   // UNICODE_TO_GBK[17326] := 16#6D0A;
   // UNICODE_TO_GBK[17327] := 16#9B96;
   // UNICODE_TO_GBK[17328] := 16#6D0B;
   // UNICODE_TO_GBK[17329] := 16#D1F3;
   // UNICODE_TO_GBK[17330] := 16#6D0C;
   // UNICODE_TO_GBK[17331] := 16#E4A3;
   // UNICODE_TO_GBK[17332] := 16#6D0D;
   // UNICODE_TO_GBK[17333] := 16#9B97;
   // UNICODE_TO_GBK[17334] := 16#6D0E;
   // UNICODE_TO_GBK[17335] := 16#E4A9;
   // UNICODE_TO_GBK[17336] := 16#6D0F;
   // UNICODE_TO_GBK[17337] := 16#9B98;
   // UNICODE_TO_GBK[17338] := 16#6D10;
   // UNICODE_TO_GBK[17339] := 16#9B99;
   // UNICODE_TO_GBK[17340] := 16#6D11;
   // UNICODE_TO_GBK[17341] := 16#9B9A;
   // UNICODE_TO_GBK[17342] := 16#6D12;
   // UNICODE_TO_GBK[17343] := 16#C8F7;
   // UNICODE_TO_GBK[17344] := 16#6D13;
   // UNICODE_TO_GBK[17345] := 16#9B9B;
   // UNICODE_TO_GBK[17346] := 16#6D14;
   // UNICODE_TO_GBK[17347] := 16#9B9C;
   // UNICODE_TO_GBK[17348] := 16#6D15;
   // UNICODE_TO_GBK[17349] := 16#9B9D;
   // UNICODE_TO_GBK[17350] := 16#6D16;
   // UNICODE_TO_GBK[17351] := 16#9B9E;
   // UNICODE_TO_GBK[17352] := 16#6D17;
   // UNICODE_TO_GBK[17353] := 16#CFB4;
   // UNICODE_TO_GBK[17354] := 16#6D18;
   // UNICODE_TO_GBK[17355] := 16#9B9F;
   // UNICODE_TO_GBK[17356] := 16#6D19;
   // UNICODE_TO_GBK[17357] := 16#E4A8;
   // UNICODE_TO_GBK[17358] := 16#6D1A;
   // UNICODE_TO_GBK[17359] := 16#E4AE;
   // UNICODE_TO_GBK[17360] := 16#6D1B;
   // UNICODE_TO_GBK[17361] := 16#C2E5;
   // UNICODE_TO_GBK[17362] := 16#6D1C;
   // UNICODE_TO_GBK[17363] := 16#9BA0;
   // UNICODE_TO_GBK[17364] := 16#6D1D;
   // UNICODE_TO_GBK[17365] := 16#9BA1;
   // UNICODE_TO_GBK[17366] := 16#6D1E;
   // UNICODE_TO_GBK[17367] := 16#B6B4;
   // UNICODE_TO_GBK[17368] := 16#6D1F;
   // UNICODE_TO_GBK[17369] := 16#9BA2;
   // UNICODE_TO_GBK[17370] := 16#6D20;
   // UNICODE_TO_GBK[17371] := 16#9BA3;
   // UNICODE_TO_GBK[17372] := 16#6D21;
   // UNICODE_TO_GBK[17373] := 16#9BA4;
   // UNICODE_TO_GBK[17374] := 16#6D22;
   // UNICODE_TO_GBK[17375] := 16#9BA5;
   // UNICODE_TO_GBK[17376] := 16#6D23;
   // UNICODE_TO_GBK[17377] := 16#9BA6;
   // UNICODE_TO_GBK[17378] := 16#6D24;
   // UNICODE_TO_GBK[17379] := 16#9BA7;
   // UNICODE_TO_GBK[17380] := 16#6D25;
   // UNICODE_TO_GBK[17381] := 16#BDF2;
   // UNICODE_TO_GBK[17382] := 16#6D26;
   // UNICODE_TO_GBK[17383] := 16#9BA8;
   // UNICODE_TO_GBK[17384] := 16#6D27;
   // UNICODE_TO_GBK[17385] := 16#E4A2;
   // UNICODE_TO_GBK[17386] := 16#6D28;
   // UNICODE_TO_GBK[17387] := 16#9BA9;
   // UNICODE_TO_GBK[17388] := 16#6D29;
   // UNICODE_TO_GBK[17389] := 16#9BAA;
   // UNICODE_TO_GBK[17390] := 16#6D2A;
   // UNICODE_TO_GBK[17391] := 16#BAE9;
   // UNICODE_TO_GBK[17392] := 16#6D2B;
   // UNICODE_TO_GBK[17393] := 16#E4AA;
   // UNICODE_TO_GBK[17394] := 16#6D2C;
   // UNICODE_TO_GBK[17395] := 16#9BAB;
   // UNICODE_TO_GBK[17396] := 16#6D2D;
   // UNICODE_TO_GBK[17397] := 16#9BAC;
   // UNICODE_TO_GBK[17398] := 16#6D2E;
   // UNICODE_TO_GBK[17399] := 16#E4AC;
   // UNICODE_TO_GBK[17400] := 16#6D2F;
   // UNICODE_TO_GBK[17401] := 16#9BAD;
   // UNICODE_TO_GBK[17402] := 16#6D30;
   // UNICODE_TO_GBK[17403] := 16#9BAE;
   // UNICODE_TO_GBK[17404] := 16#6D31;
   // UNICODE_TO_GBK[17405] := 16#B6FD;
   // UNICODE_TO_GBK[17406] := 16#6D32;
   // UNICODE_TO_GBK[17407] := 16#D6DE;
   // UNICODE_TO_GBK[17408] := 16#6D33;
   // UNICODE_TO_GBK[17409] := 16#E4B2;
   // UNICODE_TO_GBK[17410] := 16#6D34;
   // UNICODE_TO_GBK[17411] := 16#9BAF;
   // UNICODE_TO_GBK[17412] := 16#6D35;
   // UNICODE_TO_GBK[17413] := 16#E4AD;
   // UNICODE_TO_GBK[17414] := 16#6D36;
   // UNICODE_TO_GBK[17415] := 16#9BB0;
   // UNICODE_TO_GBK[17416] := 16#6D37;
   // UNICODE_TO_GBK[17417] := 16#9BB1;
   // UNICODE_TO_GBK[17418] := 16#6D38;
   // UNICODE_TO_GBK[17419] := 16#9BB2;
   // UNICODE_TO_GBK[17420] := 16#6D39;
   // UNICODE_TO_GBK[17421] := 16#E4A1;
   // UNICODE_TO_GBK[17422] := 16#6D3A;
   // UNICODE_TO_GBK[17423] := 16#9BB3;
   // UNICODE_TO_GBK[17424] := 16#6D3B;
   // UNICODE_TO_GBK[17425] := 16#BBEE;
   // UNICODE_TO_GBK[17426] := 16#6D3C;
   // UNICODE_TO_GBK[17427] := 16#CDDD;
   // UNICODE_TO_GBK[17428] := 16#6D3D;
   // UNICODE_TO_GBK[17429] := 16#C7A2;
   // UNICODE_TO_GBK[17430] := 16#6D3E;
   // UNICODE_TO_GBK[17431] := 16#C5C9;
   // UNICODE_TO_GBK[17432] := 16#6D3F;
   // UNICODE_TO_GBK[17433] := 16#9BB4;
   // UNICODE_TO_GBK[17434] := 16#6D40;
   // UNICODE_TO_GBK[17435] := 16#9BB5;
   // UNICODE_TO_GBK[17436] := 16#6D41;
   // UNICODE_TO_GBK[17437] := 16#C1F7;
   // UNICODE_TO_GBK[17438] := 16#6D42;
   // UNICODE_TO_GBK[17439] := 16#9BB6;
   // UNICODE_TO_GBK[17440] := 16#6D43;
   // UNICODE_TO_GBK[17441] := 16#E4A4;
   // UNICODE_TO_GBK[17442] := 16#6D44;
   // UNICODE_TO_GBK[17443] := 16#9BB7;
   // UNICODE_TO_GBK[17444] := 16#6D45;
   // UNICODE_TO_GBK[17445] := 16#C7B3;
   // UNICODE_TO_GBK[17446] := 16#6D46;
   // UNICODE_TO_GBK[17447] := 16#BDAC;
   // UNICODE_TO_GBK[17448] := 16#6D47;
   // UNICODE_TO_GBK[17449] := 16#BDBD;
   // UNICODE_TO_GBK[17450] := 16#6D48;
   // UNICODE_TO_GBK[17451] := 16#E4A5;
   // UNICODE_TO_GBK[17452] := 16#6D49;
   // UNICODE_TO_GBK[17453] := 16#9BB8;
   // UNICODE_TO_GBK[17454] := 16#6D4A;
   // UNICODE_TO_GBK[17455] := 16#D7C7;
   // UNICODE_TO_GBK[17456] := 16#6D4B;
   // UNICODE_TO_GBK[17457] := 16#B2E2;
   // UNICODE_TO_GBK[17458] := 16#6D4C;
   // UNICODE_TO_GBK[17459] := 16#9BB9;
   // UNICODE_TO_GBK[17460] := 16#6D4D;
   // UNICODE_TO_GBK[17461] := 16#E4AB;
   // UNICODE_TO_GBK[17462] := 16#6D4E;
   // UNICODE_TO_GBK[17463] := 16#BCC3;
   // UNICODE_TO_GBK[17464] := 16#6D4F;
   // UNICODE_TO_GBK[17465] := 16#E4AF;
   // UNICODE_TO_GBK[17466] := 16#6D50;
   // UNICODE_TO_GBK[17467] := 16#9BBA;
   // UNICODE_TO_GBK[17468] := 16#6D51;
   // UNICODE_TO_GBK[17469] := 16#BBEB;
   // UNICODE_TO_GBK[17470] := 16#6D52;
   // UNICODE_TO_GBK[17471] := 16#E4B0;
   // UNICODE_TO_GBK[17472] := 16#6D53;
   // UNICODE_TO_GBK[17473] := 16#C5A8;
   // UNICODE_TO_GBK[17474] := 16#6D54;
   // UNICODE_TO_GBK[17475] := 16#E4B1;
   // UNICODE_TO_GBK[17476] := 16#6D55;
   // UNICODE_TO_GBK[17477] := 16#9BBB;
   // UNICODE_TO_GBK[17478] := 16#6D56;
   // UNICODE_TO_GBK[17479] := 16#9BBC;
   // UNICODE_TO_GBK[17480] := 16#6D57;
   // UNICODE_TO_GBK[17481] := 16#9BBD;
   // UNICODE_TO_GBK[17482] := 16#6D58;
   // UNICODE_TO_GBK[17483] := 16#9BBE;
   // UNICODE_TO_GBK[17484] := 16#6D59;
   // UNICODE_TO_GBK[17485] := 16#D5E3;
   // UNICODE_TO_GBK[17486] := 16#6D5A;
   // UNICODE_TO_GBK[17487] := 16#BFA3;
   // UNICODE_TO_GBK[17488] := 16#6D5B;
   // UNICODE_TO_GBK[17489] := 16#9BBF;
   // UNICODE_TO_GBK[17490] := 16#6D5C;
   // UNICODE_TO_GBK[17491] := 16#E4BA;
   // UNICODE_TO_GBK[17492] := 16#6D5D;
   // UNICODE_TO_GBK[17493] := 16#9BC0;
   // UNICODE_TO_GBK[17494] := 16#6D5E;
   // UNICODE_TO_GBK[17495] := 16#E4B7;
   // UNICODE_TO_GBK[17496] := 16#6D5F;
   // UNICODE_TO_GBK[17497] := 16#9BC1;
   // UNICODE_TO_GBK[17498] := 16#6D60;
   // UNICODE_TO_GBK[17499] := 16#E4BB;
   // UNICODE_TO_GBK[17500] := 16#6D61;
   // UNICODE_TO_GBK[17501] := 16#9BC2;
   // UNICODE_TO_GBK[17502] := 16#6D62;
   // UNICODE_TO_GBK[17503] := 16#9BC3;
   // UNICODE_TO_GBK[17504] := 16#6D63;
   // UNICODE_TO_GBK[17505] := 16#E4BD;
   // UNICODE_TO_GBK[17506] := 16#6D64;
   // UNICODE_TO_GBK[17507] := 16#9BC4;
   // UNICODE_TO_GBK[17508] := 16#6D65;
   // UNICODE_TO_GBK[17509] := 16#9BC5;
   // UNICODE_TO_GBK[17510] := 16#6D66;
   // UNICODE_TO_GBK[17511] := 16#C6D6;
   // UNICODE_TO_GBK[17512] := 16#6D67;
   // UNICODE_TO_GBK[17513] := 16#9BC6;
   // UNICODE_TO_GBK[17514] := 16#6D68;
   // UNICODE_TO_GBK[17515] := 16#9BC7;
   // UNICODE_TO_GBK[17516] := 16#6D69;
   // UNICODE_TO_GBK[17517] := 16#BAC6;
   // UNICODE_TO_GBK[17518] := 16#6D6A;
   // UNICODE_TO_GBK[17519] := 16#C0CB;
   // UNICODE_TO_GBK[17520] := 16#6D6B;
   // UNICODE_TO_GBK[17521] := 16#9BC8;
   // UNICODE_TO_GBK[17522] := 16#6D6C;
   // UNICODE_TO_GBK[17523] := 16#9BC9;
   // UNICODE_TO_GBK[17524] := 16#6D6D;
   // UNICODE_TO_GBK[17525] := 16#9BCA;
   // UNICODE_TO_GBK[17526] := 16#6D6E;
   // UNICODE_TO_GBK[17527] := 16#B8A1;
   // UNICODE_TO_GBK[17528] := 16#6D6F;
   // UNICODE_TO_GBK[17529] := 16#E4B4;
   // UNICODE_TO_GBK[17530] := 16#6D70;
   // UNICODE_TO_GBK[17531] := 16#9BCB;
   // UNICODE_TO_GBK[17532] := 16#6D71;
   // UNICODE_TO_GBK[17533] := 16#9BCC;
   // UNICODE_TO_GBK[17534] := 16#6D72;
   // UNICODE_TO_GBK[17535] := 16#9BCD;
   // UNICODE_TO_GBK[17536] := 16#6D73;
   // UNICODE_TO_GBK[17537] := 16#9BCE;
   // UNICODE_TO_GBK[17538] := 16#6D74;
   // UNICODE_TO_GBK[17539] := 16#D4A1;
   // UNICODE_TO_GBK[17540] := 16#6D75;
   // UNICODE_TO_GBK[17541] := 16#9BCF;
   // UNICODE_TO_GBK[17542] := 16#6D76;
   // UNICODE_TO_GBK[17543] := 16#9BD0;
   // UNICODE_TO_GBK[17544] := 16#6D77;
   // UNICODE_TO_GBK[17545] := 16#BAA3;
   // UNICODE_TO_GBK[17546] := 16#6D78;
   // UNICODE_TO_GBK[17547] := 16#BDFE;
   // UNICODE_TO_GBK[17548] := 16#6D79;
   // UNICODE_TO_GBK[17549] := 16#9BD1;
   // UNICODE_TO_GBK[17550] := 16#6D7A;
   // UNICODE_TO_GBK[17551] := 16#9BD2;
   // UNICODE_TO_GBK[17552] := 16#6D7B;
   // UNICODE_TO_GBK[17553] := 16#9BD3;
   // UNICODE_TO_GBK[17554] := 16#6D7C;
   // UNICODE_TO_GBK[17555] := 16#E4BC;
   // UNICODE_TO_GBK[17556] := 16#6D7D;
   // UNICODE_TO_GBK[17557] := 16#9BD4;
   // UNICODE_TO_GBK[17558] := 16#6D7E;
   // UNICODE_TO_GBK[17559] := 16#9BD5;
   // UNICODE_TO_GBK[17560] := 16#6D7F;
   // UNICODE_TO_GBK[17561] := 16#9BD6;
   // UNICODE_TO_GBK[17562] := 16#6D80;
   // UNICODE_TO_GBK[17563] := 16#9BD7;
   // UNICODE_TO_GBK[17564] := 16#6D81;
   // UNICODE_TO_GBK[17565] := 16#9BD8;
   // UNICODE_TO_GBK[17566] := 16#6D82;
   // UNICODE_TO_GBK[17567] := 16#CDBF;
   // UNICODE_TO_GBK[17568] := 16#6D83;
   // UNICODE_TO_GBK[17569] := 16#9BD9;
   // UNICODE_TO_GBK[17570] := 16#6D84;
   // UNICODE_TO_GBK[17571] := 16#9BDA;
   // UNICODE_TO_GBK[17572] := 16#6D85;
   // UNICODE_TO_GBK[17573] := 16#C4F9;
   // UNICODE_TO_GBK[17574] := 16#6D86;
   // UNICODE_TO_GBK[17575] := 16#9BDB;
   // UNICODE_TO_GBK[17576] := 16#6D87;
   // UNICODE_TO_GBK[17577] := 16#9BDC;
   // UNICODE_TO_GBK[17578] := 16#6D88;
   // UNICODE_TO_GBK[17579] := 16#CFFB;
   // UNICODE_TO_GBK[17580] := 16#6D89;
   // UNICODE_TO_GBK[17581] := 16#C9E6;
   // UNICODE_TO_GBK[17582] := 16#6D8A;
   // UNICODE_TO_GBK[17583] := 16#9BDD;
   // UNICODE_TO_GBK[17584] := 16#6D8B;
   // UNICODE_TO_GBK[17585] := 16#9BDE;
   // UNICODE_TO_GBK[17586] := 16#6D8C;
   // UNICODE_TO_GBK[17587] := 16#D3BF;
   // UNICODE_TO_GBK[17588] := 16#6D8D;
   // UNICODE_TO_GBK[17589] := 16#9BDF;
   // UNICODE_TO_GBK[17590] := 16#6D8E;
   // UNICODE_TO_GBK[17591] := 16#CFD1;
   // UNICODE_TO_GBK[17592] := 16#6D8F;
   // UNICODE_TO_GBK[17593] := 16#9BE0;
   // UNICODE_TO_GBK[17594] := 16#6D90;
   // UNICODE_TO_GBK[17595] := 16#9BE1;
   // UNICODE_TO_GBK[17596] := 16#6D91;
   // UNICODE_TO_GBK[17597] := 16#E4B3;
   // UNICODE_TO_GBK[17598] := 16#6D92;
   // UNICODE_TO_GBK[17599] := 16#9BE2;
   // UNICODE_TO_GBK[17600] := 16#6D93;
   // UNICODE_TO_GBK[17601] := 16#E4B8;
   // UNICODE_TO_GBK[17602] := 16#6D94;
   // UNICODE_TO_GBK[17603] := 16#E4B9;
   // UNICODE_TO_GBK[17604] := 16#6D95;
   // UNICODE_TO_GBK[17605] := 16#CCE9;
   // UNICODE_TO_GBK[17606] := 16#6D96;
   // UNICODE_TO_GBK[17607] := 16#9BE3;
   // UNICODE_TO_GBK[17608] := 16#6D97;
   // UNICODE_TO_GBK[17609] := 16#9BE4;
   // UNICODE_TO_GBK[17610] := 16#6D98;
   // UNICODE_TO_GBK[17611] := 16#9BE5;
   // UNICODE_TO_GBK[17612] := 16#6D99;
   // UNICODE_TO_GBK[17613] := 16#9BE6;
   // UNICODE_TO_GBK[17614] := 16#6D9A;
   // UNICODE_TO_GBK[17615] := 16#9BE7;
   // UNICODE_TO_GBK[17616] := 16#6D9B;
   // UNICODE_TO_GBK[17617] := 16#CCCE;
   // UNICODE_TO_GBK[17618] := 16#6D9C;
   // UNICODE_TO_GBK[17619] := 16#9BE8;
   // UNICODE_TO_GBK[17620] := 16#6D9D;
   // UNICODE_TO_GBK[17621] := 16#C0D4;
   // UNICODE_TO_GBK[17622] := 16#6D9E;
   // UNICODE_TO_GBK[17623] := 16#E4B5;
   // UNICODE_TO_GBK[17624] := 16#6D9F;
   // UNICODE_TO_GBK[17625] := 16#C1B0;
   // UNICODE_TO_GBK[17626] := 16#6DA0;
   // UNICODE_TO_GBK[17627] := 16#E4B6;
   // UNICODE_TO_GBK[17628] := 16#6DA1;
   // UNICODE_TO_GBK[17629] := 16#CED0;
   // UNICODE_TO_GBK[17630] := 16#6DA2;
   // UNICODE_TO_GBK[17631] := 16#9BE9;
   // UNICODE_TO_GBK[17632] := 16#6DA3;
   // UNICODE_TO_GBK[17633] := 16#BBC1;
   // UNICODE_TO_GBK[17634] := 16#6DA4;
   // UNICODE_TO_GBK[17635] := 16#B5D3;
   // UNICODE_TO_GBK[17636] := 16#6DA5;
   // UNICODE_TO_GBK[17637] := 16#9BEA;
   // UNICODE_TO_GBK[17638] := 16#6DA6;
   // UNICODE_TO_GBK[17639] := 16#C8F3;
   // UNICODE_TO_GBK[17640] := 16#6DA7;
   // UNICODE_TO_GBK[17641] := 16#BDA7;
   // UNICODE_TO_GBK[17642] := 16#6DA8;
   // UNICODE_TO_GBK[17643] := 16#D5C7;
   // UNICODE_TO_GBK[17644] := 16#6DA9;
   // UNICODE_TO_GBK[17645] := 16#C9AC;
   // UNICODE_TO_GBK[17646] := 16#6DAA;
   // UNICODE_TO_GBK[17647] := 16#B8A2;
   // UNICODE_TO_GBK[17648] := 16#6DAB;
   // UNICODE_TO_GBK[17649] := 16#E4CA;
   // UNICODE_TO_GBK[17650] := 16#6DAC;
   // UNICODE_TO_GBK[17651] := 16#9BEB;
   // UNICODE_TO_GBK[17652] := 16#6DAD;
   // UNICODE_TO_GBK[17653] := 16#9BEC;
   // UNICODE_TO_GBK[17654] := 16#6DAE;
   // UNICODE_TO_GBK[17655] := 16#E4CC;
   // UNICODE_TO_GBK[17656] := 16#6DAF;
   // UNICODE_TO_GBK[17657] := 16#D1C4;
   // UNICODE_TO_GBK[17658] := 16#6DB0;
   // UNICODE_TO_GBK[17659] := 16#9BED;
   // UNICODE_TO_GBK[17660] := 16#6DB1;
   // UNICODE_TO_GBK[17661] := 16#9BEE;
   // UNICODE_TO_GBK[17662] := 16#6DB2;
   // UNICODE_TO_GBK[17663] := 16#D2BA;
   // UNICODE_TO_GBK[17664] := 16#6DB3;
   // UNICODE_TO_GBK[17665] := 16#9BEF;
   // UNICODE_TO_GBK[17666] := 16#6DB4;
   // UNICODE_TO_GBK[17667] := 16#9BF0;
   // UNICODE_TO_GBK[17668] := 16#6DB5;
   // UNICODE_TO_GBK[17669] := 16#BAAD;
   // UNICODE_TO_GBK[17670] := 16#6DB6;
   // UNICODE_TO_GBK[17671] := 16#9BF1;
   // UNICODE_TO_GBK[17672] := 16#6DB7;
   // UNICODE_TO_GBK[17673] := 16#9BF2;
   // UNICODE_TO_GBK[17674] := 16#6DB8;
   // UNICODE_TO_GBK[17675] := 16#BAD4;
   // UNICODE_TO_GBK[17676] := 16#6DB9;
   // UNICODE_TO_GBK[17677] := 16#9BF3;
   // UNICODE_TO_GBK[17678] := 16#6DBA;
   // UNICODE_TO_GBK[17679] := 16#9BF4;
   // UNICODE_TO_GBK[17680] := 16#6DBB;
   // UNICODE_TO_GBK[17681] := 16#9BF5;
   // UNICODE_TO_GBK[17682] := 16#6DBC;
   // UNICODE_TO_GBK[17683] := 16#9BF6;
   // UNICODE_TO_GBK[17684] := 16#6DBD;
   // UNICODE_TO_GBK[17685] := 16#9BF7;
   // UNICODE_TO_GBK[17686] := 16#6DBE;
   // UNICODE_TO_GBK[17687] := 16#9BF8;
   // UNICODE_TO_GBK[17688] := 16#6DBF;
   // UNICODE_TO_GBK[17689] := 16#E4C3;
   // UNICODE_TO_GBK[17690] := 16#6DC0;
   // UNICODE_TO_GBK[17691] := 16#B5ED;
   // UNICODE_TO_GBK[17692] := 16#6DC1;
   // UNICODE_TO_GBK[17693] := 16#9BF9;
   // UNICODE_TO_GBK[17694] := 16#6DC2;
   // UNICODE_TO_GBK[17695] := 16#9BFA;
   // UNICODE_TO_GBK[17696] := 16#6DC3;
   // UNICODE_TO_GBK[17697] := 16#9BFB;
   // UNICODE_TO_GBK[17698] := 16#6DC4;
   // UNICODE_TO_GBK[17699] := 16#D7CD;
   // UNICODE_TO_GBK[17700] := 16#6DC5;
   // UNICODE_TO_GBK[17701] := 16#E4C0;
   // UNICODE_TO_GBK[17702] := 16#6DC6;
   // UNICODE_TO_GBK[17703] := 16#CFFD;
   // UNICODE_TO_GBK[17704] := 16#6DC7;
   // UNICODE_TO_GBK[17705] := 16#E4BF;
   // UNICODE_TO_GBK[17706] := 16#6DC8;
   // UNICODE_TO_GBK[17707] := 16#9BFC;
   // UNICODE_TO_GBK[17708] := 16#6DC9;
   // UNICODE_TO_GBK[17709] := 16#9BFD;
   // UNICODE_TO_GBK[17710] := 16#6DCA;
   // UNICODE_TO_GBK[17711] := 16#9BFE;
   // UNICODE_TO_GBK[17712] := 16#6DCB;
   // UNICODE_TO_GBK[17713] := 16#C1DC;
   // UNICODE_TO_GBK[17714] := 16#6DCC;
   // UNICODE_TO_GBK[17715] := 16#CCCA;
   // UNICODE_TO_GBK[17716] := 16#6DCD;
   // UNICODE_TO_GBK[17717] := 16#9C40;
   // UNICODE_TO_GBK[17718] := 16#6DCE;
   // UNICODE_TO_GBK[17719] := 16#9C41;
   // UNICODE_TO_GBK[17720] := 16#6DCF;
   // UNICODE_TO_GBK[17721] := 16#9C42;
   // UNICODE_TO_GBK[17722] := 16#6DD0;
   // UNICODE_TO_GBK[17723] := 16#9C43;
   // UNICODE_TO_GBK[17724] := 16#6DD1;
   // UNICODE_TO_GBK[17725] := 16#CAE7;
   // UNICODE_TO_GBK[17726] := 16#6DD2;
   // UNICODE_TO_GBK[17727] := 16#9C44;
   // UNICODE_TO_GBK[17728] := 16#6DD3;
   // UNICODE_TO_GBK[17729] := 16#9C45;
   // UNICODE_TO_GBK[17730] := 16#6DD4;
   // UNICODE_TO_GBK[17731] := 16#9C46;
   // UNICODE_TO_GBK[17732] := 16#6DD5;
   // UNICODE_TO_GBK[17733] := 16#9C47;
   // UNICODE_TO_GBK[17734] := 16#6DD6;
   // UNICODE_TO_GBK[17735] := 16#C4D7;
   // UNICODE_TO_GBK[17736] := 16#6DD7;
   // UNICODE_TO_GBK[17737] := 16#9C48;
   // UNICODE_TO_GBK[17738] := 16#6DD8;
   // UNICODE_TO_GBK[17739] := 16#CCD4;
   // UNICODE_TO_GBK[17740] := 16#6DD9;
   // UNICODE_TO_GBK[17741] := 16#E4C8;
   // UNICODE_TO_GBK[17742] := 16#6DDA;
   // UNICODE_TO_GBK[17743] := 16#9C49;
   // UNICODE_TO_GBK[17744] := 16#6DDB;
   // UNICODE_TO_GBK[17745] := 16#9C4A;
   // UNICODE_TO_GBK[17746] := 16#6DDC;
   // UNICODE_TO_GBK[17747] := 16#9C4B;
   // UNICODE_TO_GBK[17748] := 16#6DDD;
   // UNICODE_TO_GBK[17749] := 16#E4C7;
   // UNICODE_TO_GBK[17750] := 16#6DDE;
   // UNICODE_TO_GBK[17751] := 16#E4C1;
   // UNICODE_TO_GBK[17752] := 16#6DDF;
   // UNICODE_TO_GBK[17753] := 16#9C4C;
   // UNICODE_TO_GBK[17754] := 16#6DE0;
   // UNICODE_TO_GBK[17755] := 16#E4C4;
   // UNICODE_TO_GBK[17756] := 16#6DE1;
   // UNICODE_TO_GBK[17757] := 16#B5AD;
   // UNICODE_TO_GBK[17758] := 16#6DE2;
   // UNICODE_TO_GBK[17759] := 16#9C4D;
   // UNICODE_TO_GBK[17760] := 16#6DE3;
   // UNICODE_TO_GBK[17761] := 16#9C4E;
   // UNICODE_TO_GBK[17762] := 16#6DE4;
   // UNICODE_TO_GBK[17763] := 16#D3D9;
   // UNICODE_TO_GBK[17764] := 16#6DE5;
   // UNICODE_TO_GBK[17765] := 16#9C4F;
   // UNICODE_TO_GBK[17766] := 16#6DE6;
   // UNICODE_TO_GBK[17767] := 16#E4C6;
   // UNICODE_TO_GBK[17768] := 16#6DE7;
   // UNICODE_TO_GBK[17769] := 16#9C50;
   // UNICODE_TO_GBK[17770] := 16#6DE8;
   // UNICODE_TO_GBK[17771] := 16#9C51;
   // UNICODE_TO_GBK[17772] := 16#6DE9;
   // UNICODE_TO_GBK[17773] := 16#9C52;
   // UNICODE_TO_GBK[17774] := 16#6DEA;
   // UNICODE_TO_GBK[17775] := 16#9C53;
   // UNICODE_TO_GBK[17776] := 16#6DEB;
   // UNICODE_TO_GBK[17777] := 16#D2F9;
   // UNICODE_TO_GBK[17778] := 16#6DEC;
   // UNICODE_TO_GBK[17779] := 16#B4E3;
   // UNICODE_TO_GBK[17780] := 16#6DED;
   // UNICODE_TO_GBK[17781] := 16#9C54;
   // UNICODE_TO_GBK[17782] := 16#6DEE;
   // UNICODE_TO_GBK[17783] := 16#BBB4;
   // UNICODE_TO_GBK[17784] := 16#6DEF;
   // UNICODE_TO_GBK[17785] := 16#9C55;
   // UNICODE_TO_GBK[17786] := 16#6DF0;
   // UNICODE_TO_GBK[17787] := 16#9C56;
   // UNICODE_TO_GBK[17788] := 16#6DF1;
   // UNICODE_TO_GBK[17789] := 16#C9EE;
   // UNICODE_TO_GBK[17790] := 16#6DF2;
   // UNICODE_TO_GBK[17791] := 16#9C57;
   // UNICODE_TO_GBK[17792] := 16#6DF3;
   // UNICODE_TO_GBK[17793] := 16#B4BE;
   // UNICODE_TO_GBK[17794] := 16#6DF4;
   // UNICODE_TO_GBK[17795] := 16#9C58;
   // UNICODE_TO_GBK[17796] := 16#6DF5;
   // UNICODE_TO_GBK[17797] := 16#9C59;
   // UNICODE_TO_GBK[17798] := 16#6DF6;
   // UNICODE_TO_GBK[17799] := 16#9C5A;
   // UNICODE_TO_GBK[17800] := 16#6DF7;
   // UNICODE_TO_GBK[17801] := 16#BBEC;
   // UNICODE_TO_GBK[17802] := 16#6DF8;
   // UNICODE_TO_GBK[17803] := 16#9C5B;
   // UNICODE_TO_GBK[17804] := 16#6DF9;
   // UNICODE_TO_GBK[17805] := 16#D1CD;
   // UNICODE_TO_GBK[17806] := 16#6DFA;
   // UNICODE_TO_GBK[17807] := 16#9C5C;
   // UNICODE_TO_GBK[17808] := 16#6DFB;
   // UNICODE_TO_GBK[17809] := 16#CCED;
   // UNICODE_TO_GBK[17810] := 16#6DFC;
   // UNICODE_TO_GBK[17811] := 16#EDB5;
   // UNICODE_TO_GBK[17812] := 16#6DFD;
   // UNICODE_TO_GBK[17813] := 16#9C5D;
   // UNICODE_TO_GBK[17814] := 16#6DFE;
   // UNICODE_TO_GBK[17815] := 16#9C5E;
   // UNICODE_TO_GBK[17816] := 16#6DFF;
   // UNICODE_TO_GBK[17817] := 16#9C5F;
   // UNICODE_TO_GBK[17818] := 16#6E00;
   // UNICODE_TO_GBK[17819] := 16#9C60;
   // UNICODE_TO_GBK[17820] := 16#6E01;
   // UNICODE_TO_GBK[17821] := 16#9C61;
   // UNICODE_TO_GBK[17822] := 16#6E02;
   // UNICODE_TO_GBK[17823] := 16#9C62;
   // UNICODE_TO_GBK[17824] := 16#6E03;
   // UNICODE_TO_GBK[17825] := 16#9C63;
   // UNICODE_TO_GBK[17826] := 16#6E04;
   // UNICODE_TO_GBK[17827] := 16#9C64;
   // UNICODE_TO_GBK[17828] := 16#6E05;
   // UNICODE_TO_GBK[17829] := 16#C7E5;
   // UNICODE_TO_GBK[17830] := 16#6E06;
   // UNICODE_TO_GBK[17831] := 16#9C65;
   // UNICODE_TO_GBK[17832] := 16#6E07;
   // UNICODE_TO_GBK[17833] := 16#9C66;
   // UNICODE_TO_GBK[17834] := 16#6E08;
   // UNICODE_TO_GBK[17835] := 16#9C67;
   // UNICODE_TO_GBK[17836] := 16#6E09;
   // UNICODE_TO_GBK[17837] := 16#9C68;
   // UNICODE_TO_GBK[17838] := 16#6E0A;
   // UNICODE_TO_GBK[17839] := 16#D4A8;
   // UNICODE_TO_GBK[17840] := 16#6E0B;
   // UNICODE_TO_GBK[17841] := 16#9C69;
   // UNICODE_TO_GBK[17842] := 16#6E0C;
   // UNICODE_TO_GBK[17843] := 16#E4CB;
   // UNICODE_TO_GBK[17844] := 16#6E0D;
   // UNICODE_TO_GBK[17845] := 16#D7D5;
   // UNICODE_TO_GBK[17846] := 16#6E0E;
   // UNICODE_TO_GBK[17847] := 16#E4C2;
   // UNICODE_TO_GBK[17848] := 16#6E0F;
   // UNICODE_TO_GBK[17849] := 16#9C6A;
   // UNICODE_TO_GBK[17850] := 16#6E10;
   // UNICODE_TO_GBK[17851] := 16#BDA5;
   // UNICODE_TO_GBK[17852] := 16#6E11;
   // UNICODE_TO_GBK[17853] := 16#E4C5;
   // UNICODE_TO_GBK[17854] := 16#6E12;
   // UNICODE_TO_GBK[17855] := 16#9C6B;
   // UNICODE_TO_GBK[17856] := 16#6E13;
   // UNICODE_TO_GBK[17857] := 16#9C6C;
   // UNICODE_TO_GBK[17858] := 16#6E14;
   // UNICODE_TO_GBK[17859] := 16#D3E6;
   // UNICODE_TO_GBK[17860] := 16#6E15;
   // UNICODE_TO_GBK[17861] := 16#9C6D;
   // UNICODE_TO_GBK[17862] := 16#6E16;
   // UNICODE_TO_GBK[17863] := 16#E4C9;
   // UNICODE_TO_GBK[17864] := 16#6E17;
   // UNICODE_TO_GBK[17865] := 16#C9F8;
   // UNICODE_TO_GBK[17866] := 16#6E18;
   // UNICODE_TO_GBK[17867] := 16#9C6E;
   // UNICODE_TO_GBK[17868] := 16#6E19;
   // UNICODE_TO_GBK[17869] := 16#9C6F;
   // UNICODE_TO_GBK[17870] := 16#6E1A;
   // UNICODE_TO_GBK[17871] := 16#E4BE;
   // UNICODE_TO_GBK[17872] := 16#6E1B;
   // UNICODE_TO_GBK[17873] := 16#9C70;
   // UNICODE_TO_GBK[17874] := 16#6E1C;
   // UNICODE_TO_GBK[17875] := 16#9C71;
   // UNICODE_TO_GBK[17876] := 16#6E1D;
   // UNICODE_TO_GBK[17877] := 16#D3E5;
   // UNICODE_TO_GBK[17878] := 16#6E1E;
   // UNICODE_TO_GBK[17879] := 16#9C72;
   // UNICODE_TO_GBK[17880] := 16#6E1F;
   // UNICODE_TO_GBK[17881] := 16#9C73;
   // UNICODE_TO_GBK[17882] := 16#6E20;
   // UNICODE_TO_GBK[17883] := 16#C7FE;
   // UNICODE_TO_GBK[17884] := 16#6E21;
   // UNICODE_TO_GBK[17885] := 16#B6C9;
   // UNICODE_TO_GBK[17886] := 16#6E22;
   // UNICODE_TO_GBK[17887] := 16#9C74;
   // UNICODE_TO_GBK[17888] := 16#6E23;
   // UNICODE_TO_GBK[17889] := 16#D4FC;
   // UNICODE_TO_GBK[17890] := 16#6E24;
   // UNICODE_TO_GBK[17891] := 16#B2B3;
   // UNICODE_TO_GBK[17892] := 16#6E25;
   // UNICODE_TO_GBK[17893] := 16#E4D7;
   // UNICODE_TO_GBK[17894] := 16#6E26;
   // UNICODE_TO_GBK[17895] := 16#9C75;
   // UNICODE_TO_GBK[17896] := 16#6E27;
   // UNICODE_TO_GBK[17897] := 16#9C76;
   // UNICODE_TO_GBK[17898] := 16#6E28;
   // UNICODE_TO_GBK[17899] := 16#9C77;
   // UNICODE_TO_GBK[17900] := 16#6E29;
   // UNICODE_TO_GBK[17901] := 16#CEC2;
   // UNICODE_TO_GBK[17902] := 16#6E2A;
   // UNICODE_TO_GBK[17903] := 16#9C78;
   // UNICODE_TO_GBK[17904] := 16#6E2B;
   // UNICODE_TO_GBK[17905] := 16#E4CD;
   // UNICODE_TO_GBK[17906] := 16#6E2C;
   // UNICODE_TO_GBK[17907] := 16#9C79;
   // UNICODE_TO_GBK[17908] := 16#6E2D;
   // UNICODE_TO_GBK[17909] := 16#CEBC;
   // UNICODE_TO_GBK[17910] := 16#6E2E;
   // UNICODE_TO_GBK[17911] := 16#9C7A;
   // UNICODE_TO_GBK[17912] := 16#6E2F;
   // UNICODE_TO_GBK[17913] := 16#B8DB;
   // UNICODE_TO_GBK[17914] := 16#6E30;
   // UNICODE_TO_GBK[17915] := 16#9C7B;
   // UNICODE_TO_GBK[17916] := 16#6E31;
   // UNICODE_TO_GBK[17917] := 16#9C7C;
   // UNICODE_TO_GBK[17918] := 16#6E32;
   // UNICODE_TO_GBK[17919] := 16#E4D6;
   // UNICODE_TO_GBK[17920] := 16#6E33;
   // UNICODE_TO_GBK[17921] := 16#9C7D;
   // UNICODE_TO_GBK[17922] := 16#6E34;
   // UNICODE_TO_GBK[17923] := 16#BFCA;
   // UNICODE_TO_GBK[17924] := 16#6E35;
   // UNICODE_TO_GBK[17925] := 16#9C7E;
   // UNICODE_TO_GBK[17926] := 16#6E36;
   // UNICODE_TO_GBK[17927] := 16#9C80;
   // UNICODE_TO_GBK[17928] := 16#6E37;
   // UNICODE_TO_GBK[17929] := 16#9C81;
   // UNICODE_TO_GBK[17930] := 16#6E38;
   // UNICODE_TO_GBK[17931] := 16#D3CE;
   // UNICODE_TO_GBK[17932] := 16#6E39;
   // UNICODE_TO_GBK[17933] := 16#9C82;
   // UNICODE_TO_GBK[17934] := 16#6E3A;
   // UNICODE_TO_GBK[17935] := 16#C3EC;
   // UNICODE_TO_GBK[17936] := 16#6E3B;
   // UNICODE_TO_GBK[17937] := 16#9C83;
   // UNICODE_TO_GBK[17938] := 16#6E3C;
   // UNICODE_TO_GBK[17939] := 16#9C84;
   // UNICODE_TO_GBK[17940] := 16#6E3D;
   // UNICODE_TO_GBK[17941] := 16#9C85;
   // UNICODE_TO_GBK[17942] := 16#6E3E;
   // UNICODE_TO_GBK[17943] := 16#9C86;
   // UNICODE_TO_GBK[17944] := 16#6E3F;
   // UNICODE_TO_GBK[17945] := 16#9C87;
   // UNICODE_TO_GBK[17946] := 16#6E40;
   // UNICODE_TO_GBK[17947] := 16#9C88;
   // UNICODE_TO_GBK[17948] := 16#6E41;
   // UNICODE_TO_GBK[17949] := 16#9C89;
   // UNICODE_TO_GBK[17950] := 16#6E42;
   // UNICODE_TO_GBK[17951] := 16#9C8A;
   // UNICODE_TO_GBK[17952] := 16#6E43;
   // UNICODE_TO_GBK[17953] := 16#C5C8;
   // UNICODE_TO_GBK[17954] := 16#6E44;
   // UNICODE_TO_GBK[17955] := 16#E4D8;
   // UNICODE_TO_GBK[17956] := 16#6E45;
   // UNICODE_TO_GBK[17957] := 16#9C8B;
   // UNICODE_TO_GBK[17958] := 16#6E46;
   // UNICODE_TO_GBK[17959] := 16#9C8C;
   // UNICODE_TO_GBK[17960] := 16#6E47;
   // UNICODE_TO_GBK[17961] := 16#9C8D;
   // UNICODE_TO_GBK[17962] := 16#6E48;
   // UNICODE_TO_GBK[17963] := 16#9C8E;
   // UNICODE_TO_GBK[17964] := 16#6E49;
   // UNICODE_TO_GBK[17965] := 16#9C8F;
   // UNICODE_TO_GBK[17966] := 16#6E4A;
   // UNICODE_TO_GBK[17967] := 16#9C90;
   // UNICODE_TO_GBK[17968] := 16#6E4B;
   // UNICODE_TO_GBK[17969] := 16#9C91;
   // UNICODE_TO_GBK[17970] := 16#6E4C;
   // UNICODE_TO_GBK[17971] := 16#9C92;
   // UNICODE_TO_GBK[17972] := 16#6E4D;
   // UNICODE_TO_GBK[17973] := 16#CDC4;
   // UNICODE_TO_GBK[17974] := 16#6E4E;
   // UNICODE_TO_GBK[17975] := 16#E4CF;
   // UNICODE_TO_GBK[17976] := 16#6E4F;
   // UNICODE_TO_GBK[17977] := 16#9C93;
   // UNICODE_TO_GBK[17978] := 16#6E50;
   // UNICODE_TO_GBK[17979] := 16#9C94;
   // UNICODE_TO_GBK[17980] := 16#6E51;
   // UNICODE_TO_GBK[17981] := 16#9C95;
   // UNICODE_TO_GBK[17982] := 16#6E52;
   // UNICODE_TO_GBK[17983] := 16#9C96;
   // UNICODE_TO_GBK[17984] := 16#6E53;
   // UNICODE_TO_GBK[17985] := 16#E4D4;
   // UNICODE_TO_GBK[17986] := 16#6E54;
   // UNICODE_TO_GBK[17987] := 16#E4D5;
   // UNICODE_TO_GBK[17988] := 16#6E55;
   // UNICODE_TO_GBK[17989] := 16#9C97;
   // UNICODE_TO_GBK[17990] := 16#6E56;
   // UNICODE_TO_GBK[17991] := 16#BAFE;
   // UNICODE_TO_GBK[17992] := 16#6E57;
   // UNICODE_TO_GBK[17993] := 16#9C98;
   // UNICODE_TO_GBK[17994] := 16#6E58;
   // UNICODE_TO_GBK[17995] := 16#CFE6;
   // UNICODE_TO_GBK[17996] := 16#6E59;
   // UNICODE_TO_GBK[17997] := 16#9C99;
   // UNICODE_TO_GBK[17998] := 16#6E5A;
   // UNICODE_TO_GBK[17999] := 16#9C9A;
   // UNICODE_TO_GBK[18000] := 16#6E5B;
   // UNICODE_TO_GBK[18001] := 16#D5BF;
   // UNICODE_TO_GBK[18002] := 16#6E5C;
   // UNICODE_TO_GBK[18003] := 16#9C9B;
   // UNICODE_TO_GBK[18004] := 16#6E5D;
   // UNICODE_TO_GBK[18005] := 16#9C9C;
   // UNICODE_TO_GBK[18006] := 16#6E5E;
   // UNICODE_TO_GBK[18007] := 16#9C9D;
   // UNICODE_TO_GBK[18008] := 16#6E5F;
   // UNICODE_TO_GBK[18009] := 16#E4D2;
   // UNICODE_TO_GBK[18010] := 16#6E60;
   // UNICODE_TO_GBK[18011] := 16#9C9E;
   // UNICODE_TO_GBK[18012] := 16#6E61;
   // UNICODE_TO_GBK[18013] := 16#9C9F;
   // UNICODE_TO_GBK[18014] := 16#6E62;
   // UNICODE_TO_GBK[18015] := 16#9CA0;
   // UNICODE_TO_GBK[18016] := 16#6E63;
   // UNICODE_TO_GBK[18017] := 16#9CA1;
   // UNICODE_TO_GBK[18018] := 16#6E64;
   // UNICODE_TO_GBK[18019] := 16#9CA2;
   // UNICODE_TO_GBK[18020] := 16#6E65;
   // UNICODE_TO_GBK[18021] := 16#9CA3;
   // UNICODE_TO_GBK[18022] := 16#6E66;
   // UNICODE_TO_GBK[18023] := 16#9CA4;
   // UNICODE_TO_GBK[18024] := 16#6E67;
   // UNICODE_TO_GBK[18025] := 16#9CA5;
   // UNICODE_TO_GBK[18026] := 16#6E68;
   // UNICODE_TO_GBK[18027] := 16#9CA6;
   // UNICODE_TO_GBK[18028] := 16#6E69;
   // UNICODE_TO_GBK[18029] := 16#9CA7;
   // UNICODE_TO_GBK[18030] := 16#6E6A;
   // UNICODE_TO_GBK[18031] := 16#9CA8;
   // UNICODE_TO_GBK[18032] := 16#6E6B;
   // UNICODE_TO_GBK[18033] := 16#E4D0;
   // UNICODE_TO_GBK[18034] := 16#6E6C;
   // UNICODE_TO_GBK[18035] := 16#9CA9;
   // UNICODE_TO_GBK[18036] := 16#6E6D;
   // UNICODE_TO_GBK[18037] := 16#9CAA;
   // UNICODE_TO_GBK[18038] := 16#6E6E;
   // UNICODE_TO_GBK[18039] := 16#E4CE;
   // UNICODE_TO_GBK[18040] := 16#6E6F;
   // UNICODE_TO_GBK[18041] := 16#9CAB;
   // UNICODE_TO_GBK[18042] := 16#6E70;
   // UNICODE_TO_GBK[18043] := 16#9CAC;
   // UNICODE_TO_GBK[18044] := 16#6E71;
   // UNICODE_TO_GBK[18045] := 16#9CAD;
   // UNICODE_TO_GBK[18046] := 16#6E72;
   // UNICODE_TO_GBK[18047] := 16#9CAE;
   // UNICODE_TO_GBK[18048] := 16#6E73;
   // UNICODE_TO_GBK[18049] := 16#9CAF;
   // UNICODE_TO_GBK[18050] := 16#6E74;
   // UNICODE_TO_GBK[18051] := 16#9CB0;
   // UNICODE_TO_GBK[18052] := 16#6E75;
   // UNICODE_TO_GBK[18053] := 16#9CB1;
   // UNICODE_TO_GBK[18054] := 16#6E76;
   // UNICODE_TO_GBK[18055] := 16#9CB2;
   // UNICODE_TO_GBK[18056] := 16#6E77;
   // UNICODE_TO_GBK[18057] := 16#9CB3;
   // UNICODE_TO_GBK[18058] := 16#6E78;
   // UNICODE_TO_GBK[18059] := 16#9CB4;
   // UNICODE_TO_GBK[18060] := 16#6E79;
   // UNICODE_TO_GBK[18061] := 16#9CB5;
   // UNICODE_TO_GBK[18062] := 16#6E7A;
   // UNICODE_TO_GBK[18063] := 16#9CB6;
   // UNICODE_TO_GBK[18064] := 16#6E7B;
   // UNICODE_TO_GBK[18065] := 16#9CB7;
   // UNICODE_TO_GBK[18066] := 16#6E7C;
   // UNICODE_TO_GBK[18067] := 16#9CB8;
   // UNICODE_TO_GBK[18068] := 16#6E7D;
   // UNICODE_TO_GBK[18069] := 16#9CB9;
   // UNICODE_TO_GBK[18070] := 16#6E7E;
   // UNICODE_TO_GBK[18071] := 16#CDE5;
   // UNICODE_TO_GBK[18072] := 16#6E7F;
   // UNICODE_TO_GBK[18073] := 16#CAAA;
   // UNICODE_TO_GBK[18074] := 16#6E80;
   // UNICODE_TO_GBK[18075] := 16#9CBA;
   // UNICODE_TO_GBK[18076] := 16#6E81;
   // UNICODE_TO_GBK[18077] := 16#9CBB;
   // UNICODE_TO_GBK[18078] := 16#6E82;
   // UNICODE_TO_GBK[18079] := 16#9CBC;
   // UNICODE_TO_GBK[18080] := 16#6E83;
   // UNICODE_TO_GBK[18081] := 16#C0A3;
   // UNICODE_TO_GBK[18082] := 16#6E84;
   // UNICODE_TO_GBK[18083] := 16#9CBD;
   // UNICODE_TO_GBK[18084] := 16#6E85;
   // UNICODE_TO_GBK[18085] := 16#BDA6;
   // UNICODE_TO_GBK[18086] := 16#6E86;
   // UNICODE_TO_GBK[18087] := 16#E4D3;
   // UNICODE_TO_GBK[18088] := 16#6E87;
   // UNICODE_TO_GBK[18089] := 16#9CBE;
   // UNICODE_TO_GBK[18090] := 16#6E88;
   // UNICODE_TO_GBK[18091] := 16#9CBF;
   // UNICODE_TO_GBK[18092] := 16#6E89;
   // UNICODE_TO_GBK[18093] := 16#B8C8;
   // UNICODE_TO_GBK[18094] := 16#6E8A;
   // UNICODE_TO_GBK[18095] := 16#9CC0;
   // UNICODE_TO_GBK[18096] := 16#6E8B;
   // UNICODE_TO_GBK[18097] := 16#9CC1;
   // UNICODE_TO_GBK[18098] := 16#6E8C;
   // UNICODE_TO_GBK[18099] := 16#9CC2;
   // UNICODE_TO_GBK[18100] := 16#6E8D;
   // UNICODE_TO_GBK[18101] := 16#9CC3;
   // UNICODE_TO_GBK[18102] := 16#6E8E;
   // UNICODE_TO_GBK[18103] := 16#9CC4;
   // UNICODE_TO_GBK[18104] := 16#6E8F;
   // UNICODE_TO_GBK[18105] := 16#E4E7;
   // UNICODE_TO_GBK[18106] := 16#6E90;
   // UNICODE_TO_GBK[18107] := 16#D4B4;
   // UNICODE_TO_GBK[18108] := 16#6E91;
   // UNICODE_TO_GBK[18109] := 16#9CC5;
   // UNICODE_TO_GBK[18110] := 16#6E92;
   // UNICODE_TO_GBK[18111] := 16#9CC6;
   // UNICODE_TO_GBK[18112] := 16#6E93;
   // UNICODE_TO_GBK[18113] := 16#9CC7;
   // UNICODE_TO_GBK[18114] := 16#6E94;
   // UNICODE_TO_GBK[18115] := 16#9CC8;
   // UNICODE_TO_GBK[18116] := 16#6E95;
   // UNICODE_TO_GBK[18117] := 16#9CC9;
   // UNICODE_TO_GBK[18118] := 16#6E96;
   // UNICODE_TO_GBK[18119] := 16#9CCA;
   // UNICODE_TO_GBK[18120] := 16#6E97;
   // UNICODE_TO_GBK[18121] := 16#9CCB;
   // UNICODE_TO_GBK[18122] := 16#6E98;
   // UNICODE_TO_GBK[18123] := 16#E4DB;
   // UNICODE_TO_GBK[18124] := 16#6E99;
   // UNICODE_TO_GBK[18125] := 16#9CCC;
   // UNICODE_TO_GBK[18126] := 16#6E9A;
   // UNICODE_TO_GBK[18127] := 16#9CCD;
   // UNICODE_TO_GBK[18128] := 16#6E9B;
   // UNICODE_TO_GBK[18129] := 16#9CCE;
   // UNICODE_TO_GBK[18130] := 16#6E9C;
   // UNICODE_TO_GBK[18131] := 16#C1EF;
   // UNICODE_TO_GBK[18132] := 16#6E9D;
   // UNICODE_TO_GBK[18133] := 16#9CCF;
   // UNICODE_TO_GBK[18134] := 16#6E9E;
   // UNICODE_TO_GBK[18135] := 16#9CD0;
   // UNICODE_TO_GBK[18136] := 16#6E9F;
   // UNICODE_TO_GBK[18137] := 16#E4E9;
   // UNICODE_TO_GBK[18138] := 16#6EA0;
   // UNICODE_TO_GBK[18139] := 16#9CD1;
   // UNICODE_TO_GBK[18140] := 16#6EA1;
   // UNICODE_TO_GBK[18141] := 16#9CD2;
   // UNICODE_TO_GBK[18142] := 16#6EA2;
   // UNICODE_TO_GBK[18143] := 16#D2E7;
   // UNICODE_TO_GBK[18144] := 16#6EA3;
   // UNICODE_TO_GBK[18145] := 16#9CD3;
   // UNICODE_TO_GBK[18146] := 16#6EA4;
   // UNICODE_TO_GBK[18147] := 16#9CD4;
   // UNICODE_TO_GBK[18148] := 16#6EA5;
   // UNICODE_TO_GBK[18149] := 16#E4DF;
   // UNICODE_TO_GBK[18150] := 16#6EA6;
   // UNICODE_TO_GBK[18151] := 16#9CD5;
   // UNICODE_TO_GBK[18152] := 16#6EA7;
   // UNICODE_TO_GBK[18153] := 16#E4E0;
   // UNICODE_TO_GBK[18154] := 16#6EA8;
   // UNICODE_TO_GBK[18155] := 16#9CD6;
   // UNICODE_TO_GBK[18156] := 16#6EA9;
   // UNICODE_TO_GBK[18157] := 16#9CD7;
   // UNICODE_TO_GBK[18158] := 16#6EAA;
   // UNICODE_TO_GBK[18159] := 16#CFAA;
   // UNICODE_TO_GBK[18160] := 16#6EAB;
   // UNICODE_TO_GBK[18161] := 16#9CD8;
   // UNICODE_TO_GBK[18162] := 16#6EAC;
   // UNICODE_TO_GBK[18163] := 16#9CD9;
   // UNICODE_TO_GBK[18164] := 16#6EAD;
   // UNICODE_TO_GBK[18165] := 16#9CDA;
   // UNICODE_TO_GBK[18166] := 16#6EAE;
   // UNICODE_TO_GBK[18167] := 16#9CDB;
   // UNICODE_TO_GBK[18168] := 16#6EAF;
   // UNICODE_TO_GBK[18169] := 16#CBDD;
   // UNICODE_TO_GBK[18170] := 16#6EB0;
   // UNICODE_TO_GBK[18171] := 16#9CDC;
   // UNICODE_TO_GBK[18172] := 16#6EB1;
   // UNICODE_TO_GBK[18173] := 16#E4DA;
   // UNICODE_TO_GBK[18174] := 16#6EB2;
   // UNICODE_TO_GBK[18175] := 16#E4D1;
   // UNICODE_TO_GBK[18176] := 16#6EB3;
   // UNICODE_TO_GBK[18177] := 16#9CDD;
   // UNICODE_TO_GBK[18178] := 16#6EB4;
   // UNICODE_TO_GBK[18179] := 16#E4E5;
   // UNICODE_TO_GBK[18180] := 16#6EB5;
   // UNICODE_TO_GBK[18181] := 16#9CDE;
   // UNICODE_TO_GBK[18182] := 16#6EB6;
   // UNICODE_TO_GBK[18183] := 16#C8DC;
   // UNICODE_TO_GBK[18184] := 16#6EB7;
   // UNICODE_TO_GBK[18185] := 16#E4E3;
   // UNICODE_TO_GBK[18186] := 16#6EB8;
   // UNICODE_TO_GBK[18187] := 16#9CDF;
   // UNICODE_TO_GBK[18188] := 16#6EB9;
   // UNICODE_TO_GBK[18189] := 16#9CE0;
   // UNICODE_TO_GBK[18190] := 16#6EBA;
   // UNICODE_TO_GBK[18191] := 16#C4E7;
   // UNICODE_TO_GBK[18192] := 16#6EBB;
   // UNICODE_TO_GBK[18193] := 16#E4E2;
   // UNICODE_TO_GBK[18194] := 16#6EBC;
   // UNICODE_TO_GBK[18195] := 16#9CE1;
   // UNICODE_TO_GBK[18196] := 16#6EBD;
   // UNICODE_TO_GBK[18197] := 16#E4E1;
   // UNICODE_TO_GBK[18198] := 16#6EBE;
   // UNICODE_TO_GBK[18199] := 16#9CE2;
   // UNICODE_TO_GBK[18200] := 16#6EBF;
   // UNICODE_TO_GBK[18201] := 16#9CE3;
   // UNICODE_TO_GBK[18202] := 16#6EC0;
   // UNICODE_TO_GBK[18203] := 16#9CE4;
   // UNICODE_TO_GBK[18204] := 16#6EC1;
   // UNICODE_TO_GBK[18205] := 16#B3FC;
   // UNICODE_TO_GBK[18206] := 16#6EC2;
   // UNICODE_TO_GBK[18207] := 16#E4E8;
   // UNICODE_TO_GBK[18208] := 16#6EC3;
   // UNICODE_TO_GBK[18209] := 16#9CE5;
   // UNICODE_TO_GBK[18210] := 16#6EC4;
   // UNICODE_TO_GBK[18211] := 16#9CE6;
   // UNICODE_TO_GBK[18212] := 16#6EC5;
   // UNICODE_TO_GBK[18213] := 16#9CE7;
   // UNICODE_TO_GBK[18214] := 16#6EC6;
   // UNICODE_TO_GBK[18215] := 16#9CE8;
   // UNICODE_TO_GBK[18216] := 16#6EC7;
   // UNICODE_TO_GBK[18217] := 16#B5E1;
   // UNICODE_TO_GBK[18218] := 16#6EC8;
   // UNICODE_TO_GBK[18219] := 16#9CE9;
   // UNICODE_TO_GBK[18220] := 16#6EC9;
   // UNICODE_TO_GBK[18221] := 16#9CEA;
   // UNICODE_TO_GBK[18222] := 16#6ECA;
   // UNICODE_TO_GBK[18223] := 16#9CEB;
   // UNICODE_TO_GBK[18224] := 16#6ECB;
   // UNICODE_TO_GBK[18225] := 16#D7CC;
   // UNICODE_TO_GBK[18226] := 16#6ECC;
   // UNICODE_TO_GBK[18227] := 16#9CEC;
   // UNICODE_TO_GBK[18228] := 16#6ECD;
   // UNICODE_TO_GBK[18229] := 16#9CED;
   // UNICODE_TO_GBK[18230] := 16#6ECE;
   // UNICODE_TO_GBK[18231] := 16#9CEE;
   // UNICODE_TO_GBK[18232] := 16#6ECF;
   // UNICODE_TO_GBK[18233] := 16#E4E6;
   // UNICODE_TO_GBK[18234] := 16#6ED0;
   // UNICODE_TO_GBK[18235] := 16#9CEF;
   // UNICODE_TO_GBK[18236] := 16#6ED1;
   // UNICODE_TO_GBK[18237] := 16#BBAC;
   // UNICODE_TO_GBK[18238] := 16#6ED2;
   // UNICODE_TO_GBK[18239] := 16#9CF0;
   // UNICODE_TO_GBK[18240] := 16#6ED3;
   // UNICODE_TO_GBK[18241] := 16#D7D2;
   // UNICODE_TO_GBK[18242] := 16#6ED4;
   // UNICODE_TO_GBK[18243] := 16#CCCF;
   // UNICODE_TO_GBK[18244] := 16#6ED5;
   // UNICODE_TO_GBK[18245] := 16#EBF8;
   // UNICODE_TO_GBK[18246] := 16#6ED6;
   // UNICODE_TO_GBK[18247] := 16#9CF1;
   // UNICODE_TO_GBK[18248] := 16#6ED7;
   // UNICODE_TO_GBK[18249] := 16#E4E4;
   // UNICODE_TO_GBK[18250] := 16#6ED8;
   // UNICODE_TO_GBK[18251] := 16#9CF2;
   // UNICODE_TO_GBK[18252] := 16#6ED9;
   // UNICODE_TO_GBK[18253] := 16#9CF3;
   // UNICODE_TO_GBK[18254] := 16#6EDA;
   // UNICODE_TO_GBK[18255] := 16#B9F6;
   // UNICODE_TO_GBK[18256] := 16#6EDB;
   // UNICODE_TO_GBK[18257] := 16#9CF4;
   // UNICODE_TO_GBK[18258] := 16#6EDC;
   // UNICODE_TO_GBK[18259] := 16#9CF5;
   // UNICODE_TO_GBK[18260] := 16#6EDD;
   // UNICODE_TO_GBK[18261] := 16#9CF6;
   // UNICODE_TO_GBK[18262] := 16#6EDE;
   // UNICODE_TO_GBK[18263] := 16#D6CD;
   // UNICODE_TO_GBK[18264] := 16#6EDF;
   // UNICODE_TO_GBK[18265] := 16#E4D9;
   // UNICODE_TO_GBK[18266] := 16#6EE0;
   // UNICODE_TO_GBK[18267] := 16#E4DC;
   // UNICODE_TO_GBK[18268] := 16#6EE1;
   // UNICODE_TO_GBK[18269] := 16#C2FA;
   // UNICODE_TO_GBK[18270] := 16#6EE2;
   // UNICODE_TO_GBK[18271] := 16#E4DE;
   // UNICODE_TO_GBK[18272] := 16#6EE3;
   // UNICODE_TO_GBK[18273] := 16#9CF7;
   // UNICODE_TO_GBK[18274] := 16#6EE4;
   // UNICODE_TO_GBK[18275] := 16#C2CB;
   // UNICODE_TO_GBK[18276] := 16#6EE5;
   // UNICODE_TO_GBK[18277] := 16#C0C4;
   // UNICODE_TO_GBK[18278] := 16#6EE6;
   // UNICODE_TO_GBK[18279] := 16#C2D0;
   // UNICODE_TO_GBK[18280] := 16#6EE7;
   // UNICODE_TO_GBK[18281] := 16#9CF8;
   // UNICODE_TO_GBK[18282] := 16#6EE8;
   // UNICODE_TO_GBK[18283] := 16#B1F5;
   // UNICODE_TO_GBK[18284] := 16#6EE9;
   // UNICODE_TO_GBK[18285] := 16#CCB2;
   // UNICODE_TO_GBK[18286] := 16#6EEA;
   // UNICODE_TO_GBK[18287] := 16#9CF9;
   // UNICODE_TO_GBK[18288] := 16#6EEB;
   // UNICODE_TO_GBK[18289] := 16#9CFA;
   // UNICODE_TO_GBK[18290] := 16#6EEC;
   // UNICODE_TO_GBK[18291] := 16#9CFB;
   // UNICODE_TO_GBK[18292] := 16#6EED;
   // UNICODE_TO_GBK[18293] := 16#9CFC;
   // UNICODE_TO_GBK[18294] := 16#6EEE;
   // UNICODE_TO_GBK[18295] := 16#9CFD;
   // UNICODE_TO_GBK[18296] := 16#6EEF;
   // UNICODE_TO_GBK[18297] := 16#9CFE;
   // UNICODE_TO_GBK[18298] := 16#6EF0;
   // UNICODE_TO_GBK[18299] := 16#9D40;
   // UNICODE_TO_GBK[18300] := 16#6EF1;
   // UNICODE_TO_GBK[18301] := 16#9D41;
   // UNICODE_TO_GBK[18302] := 16#6EF2;
   // UNICODE_TO_GBK[18303] := 16#9D42;
   // UNICODE_TO_GBK[18304] := 16#6EF3;
   // UNICODE_TO_GBK[18305] := 16#9D43;
   // UNICODE_TO_GBK[18306] := 16#6EF4;
   // UNICODE_TO_GBK[18307] := 16#B5CE;
   // UNICODE_TO_GBK[18308] := 16#6EF5;
   // UNICODE_TO_GBK[18309] := 16#9D44;
   // UNICODE_TO_GBK[18310] := 16#6EF6;
   // UNICODE_TO_GBK[18311] := 16#9D45;
   // UNICODE_TO_GBK[18312] := 16#6EF7;
   // UNICODE_TO_GBK[18313] := 16#9D46;
   // UNICODE_TO_GBK[18314] := 16#6EF8;
   // UNICODE_TO_GBK[18315] := 16#9D47;
   // UNICODE_TO_GBK[18316] := 16#6EF9;
   // UNICODE_TO_GBK[18317] := 16#E4EF;
   // UNICODE_TO_GBK[18318] := 16#6EFA;
   // UNICODE_TO_GBK[18319] := 16#9D48;
   // UNICODE_TO_GBK[18320] := 16#6EFB;
   // UNICODE_TO_GBK[18321] := 16#9D49;
   // UNICODE_TO_GBK[18322] := 16#6EFC;
   // UNICODE_TO_GBK[18323] := 16#9D4A;
   // UNICODE_TO_GBK[18324] := 16#6EFD;
   // UNICODE_TO_GBK[18325] := 16#9D4B;
   // UNICODE_TO_GBK[18326] := 16#6EFE;
   // UNICODE_TO_GBK[18327] := 16#9D4C;
   // UNICODE_TO_GBK[18328] := 16#6EFF;
   // UNICODE_TO_GBK[18329] := 16#9D4D;
   // UNICODE_TO_GBK[18330] := 16#6F00;
   // UNICODE_TO_GBK[18331] := 16#9D4E;
   // UNICODE_TO_GBK[18332] := 16#6F01;
   // UNICODE_TO_GBK[18333] := 16#9D4F;
   // UNICODE_TO_GBK[18334] := 16#6F02;
   // UNICODE_TO_GBK[18335] := 16#C6AF;
   // UNICODE_TO_GBK[18336] := 16#6F03;
   // UNICODE_TO_GBK[18337] := 16#9D50;
   // UNICODE_TO_GBK[18338] := 16#6F04;
   // UNICODE_TO_GBK[18339] := 16#9D51;
   // UNICODE_TO_GBK[18340] := 16#6F05;
   // UNICODE_TO_GBK[18341] := 16#9D52;
   // UNICODE_TO_GBK[18342] := 16#6F06;
   // UNICODE_TO_GBK[18343] := 16#C6E1;
   // UNICODE_TO_GBK[18344] := 16#6F07;
   // UNICODE_TO_GBK[18345] := 16#9D53;
   // UNICODE_TO_GBK[18346] := 16#6F08;
   // UNICODE_TO_GBK[18347] := 16#9D54;
   // UNICODE_TO_GBK[18348] := 16#6F09;
   // UNICODE_TO_GBK[18349] := 16#E4F5;
   // UNICODE_TO_GBK[18350] := 16#6F0A;
   // UNICODE_TO_GBK[18351] := 16#9D55;
   // UNICODE_TO_GBK[18352] := 16#6F0B;
   // UNICODE_TO_GBK[18353] := 16#9D56;
   // UNICODE_TO_GBK[18354] := 16#6F0C;
   // UNICODE_TO_GBK[18355] := 16#9D57;
   // UNICODE_TO_GBK[18356] := 16#6F0D;
   // UNICODE_TO_GBK[18357] := 16#9D58;
   // UNICODE_TO_GBK[18358] := 16#6F0E;
   // UNICODE_TO_GBK[18359] := 16#9D59;
   // UNICODE_TO_GBK[18360] := 16#6F0F;
   // UNICODE_TO_GBK[18361] := 16#C2A9;
   // UNICODE_TO_GBK[18362] := 16#6F10;
   // UNICODE_TO_GBK[18363] := 16#9D5A;
   // UNICODE_TO_GBK[18364] := 16#6F11;
   // UNICODE_TO_GBK[18365] := 16#9D5B;
   // UNICODE_TO_GBK[18366] := 16#6F12;
   // UNICODE_TO_GBK[18367] := 16#9D5C;
   // UNICODE_TO_GBK[18368] := 16#6F13;
   // UNICODE_TO_GBK[18369] := 16#C0EC;
   // UNICODE_TO_GBK[18370] := 16#6F14;
   // UNICODE_TO_GBK[18371] := 16#D1DD;
   // UNICODE_TO_GBK[18372] := 16#6F15;
   // UNICODE_TO_GBK[18373] := 16#E4EE;
   // UNICODE_TO_GBK[18374] := 16#6F16;
   // UNICODE_TO_GBK[18375] := 16#9D5D;
   // UNICODE_TO_GBK[18376] := 16#6F17;
   // UNICODE_TO_GBK[18377] := 16#9D5E;
   // UNICODE_TO_GBK[18378] := 16#6F18;
   // UNICODE_TO_GBK[18379] := 16#9D5F;
   // UNICODE_TO_GBK[18380] := 16#6F19;
   // UNICODE_TO_GBK[18381] := 16#9D60;
   // UNICODE_TO_GBK[18382] := 16#6F1A;
   // UNICODE_TO_GBK[18383] := 16#9D61;
   // UNICODE_TO_GBK[18384] := 16#6F1B;
   // UNICODE_TO_GBK[18385] := 16#9D62;
   // UNICODE_TO_GBK[18386] := 16#6F1C;
   // UNICODE_TO_GBK[18387] := 16#9D63;
   // UNICODE_TO_GBK[18388] := 16#6F1D;
   // UNICODE_TO_GBK[18389] := 16#9D64;
   // UNICODE_TO_GBK[18390] := 16#6F1E;
   // UNICODE_TO_GBK[18391] := 16#9D65;
   // UNICODE_TO_GBK[18392] := 16#6F1F;
   // UNICODE_TO_GBK[18393] := 16#9D66;
   // UNICODE_TO_GBK[18394] := 16#6F20;
   // UNICODE_TO_GBK[18395] := 16#C4AE;
   // UNICODE_TO_GBK[18396] := 16#6F21;
   // UNICODE_TO_GBK[18397] := 16#9D67;
   // UNICODE_TO_GBK[18398] := 16#6F22;
   // UNICODE_TO_GBK[18399] := 16#9D68;
   // UNICODE_TO_GBK[18400] := 16#6F23;
   // UNICODE_TO_GBK[18401] := 16#9D69;
   // UNICODE_TO_GBK[18402] := 16#6F24;
   // UNICODE_TO_GBK[18403] := 16#E4ED;
   // UNICODE_TO_GBK[18404] := 16#6F25;
   // UNICODE_TO_GBK[18405] := 16#9D6A;
   // UNICODE_TO_GBK[18406] := 16#6F26;
   // UNICODE_TO_GBK[18407] := 16#9D6B;
   // UNICODE_TO_GBK[18408] := 16#6F27;
   // UNICODE_TO_GBK[18409] := 16#9D6C;
   // UNICODE_TO_GBK[18410] := 16#6F28;
   // UNICODE_TO_GBK[18411] := 16#9D6D;
   // UNICODE_TO_GBK[18412] := 16#6F29;
   // UNICODE_TO_GBK[18413] := 16#E4F6;
   // UNICODE_TO_GBK[18414] := 16#6F2A;
   // UNICODE_TO_GBK[18415] := 16#E4F4;
   // UNICODE_TO_GBK[18416] := 16#6F2B;
   // UNICODE_TO_GBK[18417] := 16#C2FE;
   // UNICODE_TO_GBK[18418] := 16#6F2C;
   // UNICODE_TO_GBK[18419] := 16#9D6E;
   // UNICODE_TO_GBK[18420] := 16#6F2D;
   // UNICODE_TO_GBK[18421] := 16#E4DD;
   // UNICODE_TO_GBK[18422] := 16#6F2E;
   // UNICODE_TO_GBK[18423] := 16#9D6F;
   // UNICODE_TO_GBK[18424] := 16#6F2F;
   // UNICODE_TO_GBK[18425] := 16#E4F0;
   // UNICODE_TO_GBK[18426] := 16#6F30;
   // UNICODE_TO_GBK[18427] := 16#9D70;
   // UNICODE_TO_GBK[18428] := 16#6F31;
   // UNICODE_TO_GBK[18429] := 16#CAFE;
   // UNICODE_TO_GBK[18430] := 16#6F32;
   // UNICODE_TO_GBK[18431] := 16#9D71;
   // UNICODE_TO_GBK[18432] := 16#6F33;
   // UNICODE_TO_GBK[18433] := 16#D5C4;
   // UNICODE_TO_GBK[18434] := 16#6F34;
   // UNICODE_TO_GBK[18435] := 16#9D72;
   // UNICODE_TO_GBK[18436] := 16#6F35;
   // UNICODE_TO_GBK[18437] := 16#9D73;
   // UNICODE_TO_GBK[18438] := 16#6F36;
   // UNICODE_TO_GBK[18439] := 16#E4F1;
   // UNICODE_TO_GBK[18440] := 16#6F37;
   // UNICODE_TO_GBK[18441] := 16#9D74;
   // UNICODE_TO_GBK[18442] := 16#6F38;
   // UNICODE_TO_GBK[18443] := 16#9D75;
   // UNICODE_TO_GBK[18444] := 16#6F39;
   // UNICODE_TO_GBK[18445] := 16#9D76;
   // UNICODE_TO_GBK[18446] := 16#6F3A;
   // UNICODE_TO_GBK[18447] := 16#9D77;
   // UNICODE_TO_GBK[18448] := 16#6F3B;
   // UNICODE_TO_GBK[18449] := 16#9D78;
   // UNICODE_TO_GBK[18450] := 16#6F3C;
   // UNICODE_TO_GBK[18451] := 16#9D79;
   // UNICODE_TO_GBK[18452] := 16#6F3D;
   // UNICODE_TO_GBK[18453] := 16#9D7A;
   // UNICODE_TO_GBK[18454] := 16#6F3E;
   // UNICODE_TO_GBK[18455] := 16#D1FA;
   // UNICODE_TO_GBK[18456] := 16#6F3F;
   // UNICODE_TO_GBK[18457] := 16#9D7B;
   // UNICODE_TO_GBK[18458] := 16#6F40;
   // UNICODE_TO_GBK[18459] := 16#9D7C;
   // UNICODE_TO_GBK[18460] := 16#6F41;
   // UNICODE_TO_GBK[18461] := 16#9D7D;
   // UNICODE_TO_GBK[18462] := 16#6F42;
   // UNICODE_TO_GBK[18463] := 16#9D7E;
   // UNICODE_TO_GBK[18464] := 16#6F43;
   // UNICODE_TO_GBK[18465] := 16#9D80;
   // UNICODE_TO_GBK[18466] := 16#6F44;
   // UNICODE_TO_GBK[18467] := 16#9D81;
   // UNICODE_TO_GBK[18468] := 16#6F45;
   // UNICODE_TO_GBK[18469] := 16#9D82;
   // UNICODE_TO_GBK[18470] := 16#6F46;
   // UNICODE_TO_GBK[18471] := 16#E4EB;
   // UNICODE_TO_GBK[18472] := 16#6F47;
   // UNICODE_TO_GBK[18473] := 16#E4EC;
   // UNICODE_TO_GBK[18474] := 16#6F48;
   // UNICODE_TO_GBK[18475] := 16#9D83;
   // UNICODE_TO_GBK[18476] := 16#6F49;
   // UNICODE_TO_GBK[18477] := 16#9D84;
   // UNICODE_TO_GBK[18478] := 16#6F4A;
   // UNICODE_TO_GBK[18479] := 16#9D85;
   // UNICODE_TO_GBK[18480] := 16#6F4B;
   // UNICODE_TO_GBK[18481] := 16#E4F2;
   // UNICODE_TO_GBK[18482] := 16#6F4C;
   // UNICODE_TO_GBK[18483] := 16#9D86;
   // UNICODE_TO_GBK[18484] := 16#6F4D;
   // UNICODE_TO_GBK[18485] := 16#CEAB;
   // UNICODE_TO_GBK[18486] := 16#6F4E;
   // UNICODE_TO_GBK[18487] := 16#9D87;
   // UNICODE_TO_GBK[18488] := 16#6F4F;
   // UNICODE_TO_GBK[18489] := 16#9D88;
   // UNICODE_TO_GBK[18490] := 16#6F50;
   // UNICODE_TO_GBK[18491] := 16#9D89;
   // UNICODE_TO_GBK[18492] := 16#6F51;
   // UNICODE_TO_GBK[18493] := 16#9D8A;
   // UNICODE_TO_GBK[18494] := 16#6F52;
   // UNICODE_TO_GBK[18495] := 16#9D8B;
   // UNICODE_TO_GBK[18496] := 16#6F53;
   // UNICODE_TO_GBK[18497] := 16#9D8C;
   // UNICODE_TO_GBK[18498] := 16#6F54;
   // UNICODE_TO_GBK[18499] := 16#9D8D;
   // UNICODE_TO_GBK[18500] := 16#6F55;
   // UNICODE_TO_GBK[18501] := 16#9D8E;
   // UNICODE_TO_GBK[18502] := 16#6F56;
   // UNICODE_TO_GBK[18503] := 16#9D8F;
   // UNICODE_TO_GBK[18504] := 16#6F57;
   // UNICODE_TO_GBK[18505] := 16#9D90;
   // UNICODE_TO_GBK[18506] := 16#6F58;
   // UNICODE_TO_GBK[18507] := 16#C5CB;
   // UNICODE_TO_GBK[18508] := 16#6F59;
   // UNICODE_TO_GBK[18509] := 16#9D91;
   // UNICODE_TO_GBK[18510] := 16#6F5A;
   // UNICODE_TO_GBK[18511] := 16#9D92;
   // UNICODE_TO_GBK[18512] := 16#6F5B;
   // UNICODE_TO_GBK[18513] := 16#9D93;
   // UNICODE_TO_GBK[18514] := 16#6F5C;
   // UNICODE_TO_GBK[18515] := 16#C7B1;
   // UNICODE_TO_GBK[18516] := 16#6F5D;
   // UNICODE_TO_GBK[18517] := 16#9D94;
   // UNICODE_TO_GBK[18518] := 16#6F5E;
   // UNICODE_TO_GBK[18519] := 16#C2BA;
   // UNICODE_TO_GBK[18520] := 16#6F5F;
   // UNICODE_TO_GBK[18521] := 16#9D95;
   // UNICODE_TO_GBK[18522] := 16#6F60;
   // UNICODE_TO_GBK[18523] := 16#9D96;
   // UNICODE_TO_GBK[18524] := 16#6F61;
   // UNICODE_TO_GBK[18525] := 16#9D97;
   // UNICODE_TO_GBK[18526] := 16#6F62;
   // UNICODE_TO_GBK[18527] := 16#E4EA;
   // UNICODE_TO_GBK[18528] := 16#6F63;
   // UNICODE_TO_GBK[18529] := 16#9D98;
   // UNICODE_TO_GBK[18530] := 16#6F64;
   // UNICODE_TO_GBK[18531] := 16#9D99;
   // UNICODE_TO_GBK[18532] := 16#6F65;
   // UNICODE_TO_GBK[18533] := 16#9D9A;
   // UNICODE_TO_GBK[18534] := 16#6F66;
   // UNICODE_TO_GBK[18535] := 16#C1CA;
   // UNICODE_TO_GBK[18536] := 16#6F67;
   // UNICODE_TO_GBK[18537] := 16#9D9B;
   // UNICODE_TO_GBK[18538] := 16#6F68;
   // UNICODE_TO_GBK[18539] := 16#9D9C;
   // UNICODE_TO_GBK[18540] := 16#6F69;
   // UNICODE_TO_GBK[18541] := 16#9D9D;
   // UNICODE_TO_GBK[18542] := 16#6F6A;
   // UNICODE_TO_GBK[18543] := 16#9D9E;
   // UNICODE_TO_GBK[18544] := 16#6F6B;
   // UNICODE_TO_GBK[18545] := 16#9D9F;
   // UNICODE_TO_GBK[18546] := 16#6F6C;
   // UNICODE_TO_GBK[18547] := 16#9DA0;
   // UNICODE_TO_GBK[18548] := 16#6F6D;
   // UNICODE_TO_GBK[18549] := 16#CCB6;
   // UNICODE_TO_GBK[18550] := 16#6F6E;
   // UNICODE_TO_GBK[18551] := 16#B3B1;
   // UNICODE_TO_GBK[18552] := 16#6F6F;
   // UNICODE_TO_GBK[18553] := 16#9DA1;
   // UNICODE_TO_GBK[18554] := 16#6F70;
   // UNICODE_TO_GBK[18555] := 16#9DA2;
   // UNICODE_TO_GBK[18556] := 16#6F71;
   // UNICODE_TO_GBK[18557] := 16#9DA3;
   // UNICODE_TO_GBK[18558] := 16#6F72;
   // UNICODE_TO_GBK[18559] := 16#E4FB;
   // UNICODE_TO_GBK[18560] := 16#6F73;
   // UNICODE_TO_GBK[18561] := 16#9DA4;
   // UNICODE_TO_GBK[18562] := 16#6F74;
   // UNICODE_TO_GBK[18563] := 16#E4F3;
   // UNICODE_TO_GBK[18564] := 16#6F75;
   // UNICODE_TO_GBK[18565] := 16#9DA5;
   // UNICODE_TO_GBK[18566] := 16#6F76;
   // UNICODE_TO_GBK[18567] := 16#9DA6;
   // UNICODE_TO_GBK[18568] := 16#6F77;
   // UNICODE_TO_GBK[18569] := 16#9DA7;
   // UNICODE_TO_GBK[18570] := 16#6F78;
   // UNICODE_TO_GBK[18571] := 16#E4FA;
   // UNICODE_TO_GBK[18572] := 16#6F79;
   // UNICODE_TO_GBK[18573] := 16#9DA8;
   // UNICODE_TO_GBK[18574] := 16#6F7A;
   // UNICODE_TO_GBK[18575] := 16#E4FD;
   // UNICODE_TO_GBK[18576] := 16#6F7B;
   // UNICODE_TO_GBK[18577] := 16#9DA9;
   // UNICODE_TO_GBK[18578] := 16#6F7C;
   // UNICODE_TO_GBK[18579] := 16#E4FC;
   // UNICODE_TO_GBK[18580] := 16#6F7D;
   // UNICODE_TO_GBK[18581] := 16#9DAA;
   // UNICODE_TO_GBK[18582] := 16#6F7E;
   // UNICODE_TO_GBK[18583] := 16#9DAB;
   // UNICODE_TO_GBK[18584] := 16#6F7F;
   // UNICODE_TO_GBK[18585] := 16#9DAC;
   // UNICODE_TO_GBK[18586] := 16#6F80;
   // UNICODE_TO_GBK[18587] := 16#9DAD;
   // UNICODE_TO_GBK[18588] := 16#6F81;
   // UNICODE_TO_GBK[18589] := 16#9DAE;
   // UNICODE_TO_GBK[18590] := 16#6F82;
   // UNICODE_TO_GBK[18591] := 16#9DAF;
   // UNICODE_TO_GBK[18592] := 16#6F83;
   // UNICODE_TO_GBK[18593] := 16#9DB0;
   // UNICODE_TO_GBK[18594] := 16#6F84;
   // UNICODE_TO_GBK[18595] := 16#B3CE;
   // UNICODE_TO_GBK[18596] := 16#6F85;
   // UNICODE_TO_GBK[18597] := 16#9DB1;
   // UNICODE_TO_GBK[18598] := 16#6F86;
   // UNICODE_TO_GBK[18599] := 16#9DB2;
   // UNICODE_TO_GBK[18600] := 16#6F87;
   // UNICODE_TO_GBK[18601] := 16#9DB3;
   // UNICODE_TO_GBK[18602] := 16#6F88;
   // UNICODE_TO_GBK[18603] := 16#B3BA;
   // UNICODE_TO_GBK[18604] := 16#6F89;
   // UNICODE_TO_GBK[18605] := 16#E4F7;
   // UNICODE_TO_GBK[18606] := 16#6F8A;
   // UNICODE_TO_GBK[18607] := 16#9DB4;
   // UNICODE_TO_GBK[18608] := 16#6F8B;
   // UNICODE_TO_GBK[18609] := 16#9DB5;
   // UNICODE_TO_GBK[18610] := 16#6F8C;
   // UNICODE_TO_GBK[18611] := 16#E4F9;
   // UNICODE_TO_GBK[18612] := 16#6F8D;
   // UNICODE_TO_GBK[18613] := 16#E4F8;
   // UNICODE_TO_GBK[18614] := 16#6F8E;
   // UNICODE_TO_GBK[18615] := 16#C5EC;
   // UNICODE_TO_GBK[18616] := 16#6F8F;
   // UNICODE_TO_GBK[18617] := 16#9DB6;
   // UNICODE_TO_GBK[18618] := 16#6F90;
   // UNICODE_TO_GBK[18619] := 16#9DB7;
   // UNICODE_TO_GBK[18620] := 16#6F91;
   // UNICODE_TO_GBK[18621] := 16#9DB8;
   // UNICODE_TO_GBK[18622] := 16#6F92;
   // UNICODE_TO_GBK[18623] := 16#9DB9;
   // UNICODE_TO_GBK[18624] := 16#6F93;
   // UNICODE_TO_GBK[18625] := 16#9DBA;
   // UNICODE_TO_GBK[18626] := 16#6F94;
   // UNICODE_TO_GBK[18627] := 16#9DBB;
   // UNICODE_TO_GBK[18628] := 16#6F95;
   // UNICODE_TO_GBK[18629] := 16#9DBC;
   // UNICODE_TO_GBK[18630] := 16#6F96;
   // UNICODE_TO_GBK[18631] := 16#9DBD;
   // UNICODE_TO_GBK[18632] := 16#6F97;
   // UNICODE_TO_GBK[18633] := 16#9DBE;
   // UNICODE_TO_GBK[18634] := 16#6F98;
   // UNICODE_TO_GBK[18635] := 16#9DBF;
   // UNICODE_TO_GBK[18636] := 16#6F99;
   // UNICODE_TO_GBK[18637] := 16#9DC0;
   // UNICODE_TO_GBK[18638] := 16#6F9A;
   // UNICODE_TO_GBK[18639] := 16#9DC1;
   // UNICODE_TO_GBK[18640] := 16#6F9B;
   // UNICODE_TO_GBK[18641] := 16#9DC2;
   // UNICODE_TO_GBK[18642] := 16#6F9C;
   // UNICODE_TO_GBK[18643] := 16#C0BD;
   // UNICODE_TO_GBK[18644] := 16#6F9D;
   // UNICODE_TO_GBK[18645] := 16#9DC3;
   // UNICODE_TO_GBK[18646] := 16#6F9E;
   // UNICODE_TO_GBK[18647] := 16#9DC4;
   // UNICODE_TO_GBK[18648] := 16#6F9F;
   // UNICODE_TO_GBK[18649] := 16#9DC5;
   // UNICODE_TO_GBK[18650] := 16#6FA0;
   // UNICODE_TO_GBK[18651] := 16#9DC6;
   // UNICODE_TO_GBK[18652] := 16#6FA1;
   // UNICODE_TO_GBK[18653] := 16#D4E8;
   // UNICODE_TO_GBK[18654] := 16#6FA2;
   // UNICODE_TO_GBK[18655] := 16#9DC7;
   // UNICODE_TO_GBK[18656] := 16#6FA3;
   // UNICODE_TO_GBK[18657] := 16#9DC8;
   // UNICODE_TO_GBK[18658] := 16#6FA4;
   // UNICODE_TO_GBK[18659] := 16#9DC9;
   // UNICODE_TO_GBK[18660] := 16#6FA5;
   // UNICODE_TO_GBK[18661] := 16#9DCA;
   // UNICODE_TO_GBK[18662] := 16#6FA6;
   // UNICODE_TO_GBK[18663] := 16#9DCB;
   // UNICODE_TO_GBK[18664] := 16#6FA7;
   // UNICODE_TO_GBK[18665] := 16#E5A2;
   // UNICODE_TO_GBK[18666] := 16#6FA8;
   // UNICODE_TO_GBK[18667] := 16#9DCC;
   // UNICODE_TO_GBK[18668] := 16#6FA9;
   // UNICODE_TO_GBK[18669] := 16#9DCD;
   // UNICODE_TO_GBK[18670] := 16#6FAA;
   // UNICODE_TO_GBK[18671] := 16#9DCE;
   // UNICODE_TO_GBK[18672] := 16#6FAB;
   // UNICODE_TO_GBK[18673] := 16#9DCF;
   // UNICODE_TO_GBK[18674] := 16#6FAC;
   // UNICODE_TO_GBK[18675] := 16#9DD0;
   // UNICODE_TO_GBK[18676] := 16#6FAD;
   // UNICODE_TO_GBK[18677] := 16#9DD1;
   // UNICODE_TO_GBK[18678] := 16#6FAE;
   // UNICODE_TO_GBK[18679] := 16#9DD2;
   // UNICODE_TO_GBK[18680] := 16#6FAF;
   // UNICODE_TO_GBK[18681] := 16#9DD3;
   // UNICODE_TO_GBK[18682] := 16#6FB0;
   // UNICODE_TO_GBK[18683] := 16#9DD4;
   // UNICODE_TO_GBK[18684] := 16#6FB1;
   // UNICODE_TO_GBK[18685] := 16#9DD5;
   // UNICODE_TO_GBK[18686] := 16#6FB2;
   // UNICODE_TO_GBK[18687] := 16#9DD6;
   // UNICODE_TO_GBK[18688] := 16#6FB3;
   // UNICODE_TO_GBK[18689] := 16#B0C4;
   // UNICODE_TO_GBK[18690] := 16#6FB4;
   // UNICODE_TO_GBK[18691] := 16#9DD7;
   // UNICODE_TO_GBK[18692] := 16#6FB5;
   // UNICODE_TO_GBK[18693] := 16#9DD8;
   // UNICODE_TO_GBK[18694] := 16#6FB6;
   // UNICODE_TO_GBK[18695] := 16#E5A4;
   // UNICODE_TO_GBK[18696] := 16#6FB7;
   // UNICODE_TO_GBK[18697] := 16#9DD9;
   // UNICODE_TO_GBK[18698] := 16#6FB8;
   // UNICODE_TO_GBK[18699] := 16#9DDA;
   // UNICODE_TO_GBK[18700] := 16#6FB9;
   // UNICODE_TO_GBK[18701] := 16#E5A3;
   // UNICODE_TO_GBK[18702] := 16#6FBA;
   // UNICODE_TO_GBK[18703] := 16#9DDB;
   // UNICODE_TO_GBK[18704] := 16#6FBB;
   // UNICODE_TO_GBK[18705] := 16#9DDC;
   // UNICODE_TO_GBK[18706] := 16#6FBC;
   // UNICODE_TO_GBK[18707] := 16#9DDD;
   // UNICODE_TO_GBK[18708] := 16#6FBD;
   // UNICODE_TO_GBK[18709] := 16#9DDE;
   // UNICODE_TO_GBK[18710] := 16#6FBE;
   // UNICODE_TO_GBK[18711] := 16#9DDF;
   // UNICODE_TO_GBK[18712] := 16#6FBF;
   // UNICODE_TO_GBK[18713] := 16#9DE0;
   // UNICODE_TO_GBK[18714] := 16#6FC0;
   // UNICODE_TO_GBK[18715] := 16#BCA4;
   // UNICODE_TO_GBK[18716] := 16#6FC1;
   // UNICODE_TO_GBK[18717] := 16#9DE1;
   // UNICODE_TO_GBK[18718] := 16#6FC2;
   // UNICODE_TO_GBK[18719] := 16#E5A5;
   // UNICODE_TO_GBK[18720] := 16#6FC3;
   // UNICODE_TO_GBK[18721] := 16#9DE2;
   // UNICODE_TO_GBK[18722] := 16#6FC4;
   // UNICODE_TO_GBK[18723] := 16#9DE3;
   // UNICODE_TO_GBK[18724] := 16#6FC5;
   // UNICODE_TO_GBK[18725] := 16#9DE4;
   // UNICODE_TO_GBK[18726] := 16#6FC6;
   // UNICODE_TO_GBK[18727] := 16#9DE5;
   // UNICODE_TO_GBK[18728] := 16#6FC7;
   // UNICODE_TO_GBK[18729] := 16#9DE6;
   // UNICODE_TO_GBK[18730] := 16#6FC8;
   // UNICODE_TO_GBK[18731] := 16#9DE7;
   // UNICODE_TO_GBK[18732] := 16#6FC9;
   // UNICODE_TO_GBK[18733] := 16#E5A1;
   // UNICODE_TO_GBK[18734] := 16#6FCA;
   // UNICODE_TO_GBK[18735] := 16#9DE8;
   // UNICODE_TO_GBK[18736] := 16#6FCB;
   // UNICODE_TO_GBK[18737] := 16#9DE9;
   // UNICODE_TO_GBK[18738] := 16#6FCC;
   // UNICODE_TO_GBK[18739] := 16#9DEA;
   // UNICODE_TO_GBK[18740] := 16#6FCD;
   // UNICODE_TO_GBK[18741] := 16#9DEB;
   // UNICODE_TO_GBK[18742] := 16#6FCE;
   // UNICODE_TO_GBK[18743] := 16#9DEC;
   // UNICODE_TO_GBK[18744] := 16#6FCF;
   // UNICODE_TO_GBK[18745] := 16#9DED;
   // UNICODE_TO_GBK[18746] := 16#6FD0;
   // UNICODE_TO_GBK[18747] := 16#9DEE;
   // UNICODE_TO_GBK[18748] := 16#6FD1;
   // UNICODE_TO_GBK[18749] := 16#E4FE;
   // UNICODE_TO_GBK[18750] := 16#6FD2;
   // UNICODE_TO_GBK[18751] := 16#B1F4;
   // UNICODE_TO_GBK[18752] := 16#6FD3;
   // UNICODE_TO_GBK[18753] := 16#9DEF;
   // UNICODE_TO_GBK[18754] := 16#6FD4;
   // UNICODE_TO_GBK[18755] := 16#9DF0;
   // UNICODE_TO_GBK[18756] := 16#6FD5;
   // UNICODE_TO_GBK[18757] := 16#9DF1;
   // UNICODE_TO_GBK[18758] := 16#6FD6;
   // UNICODE_TO_GBK[18759] := 16#9DF2;
   // UNICODE_TO_GBK[18760] := 16#6FD7;
   // UNICODE_TO_GBK[18761] := 16#9DF3;
   // UNICODE_TO_GBK[18762] := 16#6FD8;
   // UNICODE_TO_GBK[18763] := 16#9DF4;
   // UNICODE_TO_GBK[18764] := 16#6FD9;
   // UNICODE_TO_GBK[18765] := 16#9DF5;
   // UNICODE_TO_GBK[18766] := 16#6FDA;
   // UNICODE_TO_GBK[18767] := 16#9DF6;
   // UNICODE_TO_GBK[18768] := 16#6FDB;
   // UNICODE_TO_GBK[18769] := 16#9DF7;
   // UNICODE_TO_GBK[18770] := 16#6FDC;
   // UNICODE_TO_GBK[18771] := 16#9DF8;
   // UNICODE_TO_GBK[18772] := 16#6FDD;
   // UNICODE_TO_GBK[18773] := 16#9DF9;
   // UNICODE_TO_GBK[18774] := 16#6FDE;
   // UNICODE_TO_GBK[18775] := 16#E5A8;
   // UNICODE_TO_GBK[18776] := 16#6FDF;
   // UNICODE_TO_GBK[18777] := 16#9DFA;
   // UNICODE_TO_GBK[18778] := 16#6FE0;
   // UNICODE_TO_GBK[18779] := 16#E5A9;
   // UNICODE_TO_GBK[18780] := 16#6FE1;
   // UNICODE_TO_GBK[18781] := 16#E5A6;
   // UNICODE_TO_GBK[18782] := 16#6FE2;
   // UNICODE_TO_GBK[18783] := 16#9DFB;
   // UNICODE_TO_GBK[18784] := 16#6FE3;
   // UNICODE_TO_GBK[18785] := 16#9DFC;
   // UNICODE_TO_GBK[18786] := 16#6FE4;
   // UNICODE_TO_GBK[18787] := 16#9DFD;
   // UNICODE_TO_GBK[18788] := 16#6FE5;
   // UNICODE_TO_GBK[18789] := 16#9DFE;
   // UNICODE_TO_GBK[18790] := 16#6FE6;
   // UNICODE_TO_GBK[18791] := 16#9E40;
   // UNICODE_TO_GBK[18792] := 16#6FE7;
   // UNICODE_TO_GBK[18793] := 16#9E41;
   // UNICODE_TO_GBK[18794] := 16#6FE8;
   // UNICODE_TO_GBK[18795] := 16#9E42;
   // UNICODE_TO_GBK[18796] := 16#6FE9;
   // UNICODE_TO_GBK[18797] := 16#9E43;
   // UNICODE_TO_GBK[18798] := 16#6FEA;
   // UNICODE_TO_GBK[18799] := 16#9E44;
   // UNICODE_TO_GBK[18800] := 16#6FEB;
   // UNICODE_TO_GBK[18801] := 16#9E45;
   // UNICODE_TO_GBK[18802] := 16#6FEC;
   // UNICODE_TO_GBK[18803] := 16#9E46;
   // UNICODE_TO_GBK[18804] := 16#6FED;
   // UNICODE_TO_GBK[18805] := 16#9E47;
   // UNICODE_TO_GBK[18806] := 16#6FEE;
   // UNICODE_TO_GBK[18807] := 16#E5A7;
   // UNICODE_TO_GBK[18808] := 16#6FEF;
   // UNICODE_TO_GBK[18809] := 16#E5AA;
   // UNICODE_TO_GBK[18810] := 16#6FF0;
   // UNICODE_TO_GBK[18811] := 16#9E48;
   // UNICODE_TO_GBK[18812] := 16#6FF1;
   // UNICODE_TO_GBK[18813] := 16#9E49;
   // UNICODE_TO_GBK[18814] := 16#6FF2;
   // UNICODE_TO_GBK[18815] := 16#9E4A;
   // UNICODE_TO_GBK[18816] := 16#6FF3;
   // UNICODE_TO_GBK[18817] := 16#9E4B;
   // UNICODE_TO_GBK[18818] := 16#6FF4;
   // UNICODE_TO_GBK[18819] := 16#9E4C;
   // UNICODE_TO_GBK[18820] := 16#6FF5;
   // UNICODE_TO_GBK[18821] := 16#9E4D;
   // UNICODE_TO_GBK[18822] := 16#6FF6;
   // UNICODE_TO_GBK[18823] := 16#9E4E;
   // UNICODE_TO_GBK[18824] := 16#6FF7;
   // UNICODE_TO_GBK[18825] := 16#9E4F;
   // UNICODE_TO_GBK[18826] := 16#6FF8;
   // UNICODE_TO_GBK[18827] := 16#9E50;
   // UNICODE_TO_GBK[18828] := 16#6FF9;
   // UNICODE_TO_GBK[18829] := 16#9E51;
   // UNICODE_TO_GBK[18830] := 16#6FFA;
   // UNICODE_TO_GBK[18831] := 16#9E52;
   // UNICODE_TO_GBK[18832] := 16#6FFB;
   // UNICODE_TO_GBK[18833] := 16#9E53;
   // UNICODE_TO_GBK[18834] := 16#6FFC;
   // UNICODE_TO_GBK[18835] := 16#9E54;
   // UNICODE_TO_GBK[18836] := 16#6FFD;
   // UNICODE_TO_GBK[18837] := 16#9E55;
   // UNICODE_TO_GBK[18838] := 16#6FFE;
   // UNICODE_TO_GBK[18839] := 16#9E56;
   // UNICODE_TO_GBK[18840] := 16#6FFF;
   // UNICODE_TO_GBK[18841] := 16#9E57;
   // UNICODE_TO_GBK[18842] := 16#7000;
   // UNICODE_TO_GBK[18843] := 16#9E58;
   // UNICODE_TO_GBK[18844] := 16#7001;
   // UNICODE_TO_GBK[18845] := 16#9E59;
   // UNICODE_TO_GBK[18846] := 16#7002;
   // UNICODE_TO_GBK[18847] := 16#9E5A;
   // UNICODE_TO_GBK[18848] := 16#7003;
   // UNICODE_TO_GBK[18849] := 16#9E5B;
   // UNICODE_TO_GBK[18850] := 16#7004;
   // UNICODE_TO_GBK[18851] := 16#9E5C;
   // UNICODE_TO_GBK[18852] := 16#7005;
   // UNICODE_TO_GBK[18853] := 16#9E5D;
   // UNICODE_TO_GBK[18854] := 16#7006;
   // UNICODE_TO_GBK[18855] := 16#9E5E;
   // UNICODE_TO_GBK[18856] := 16#7007;
   // UNICODE_TO_GBK[18857] := 16#9E5F;
   // UNICODE_TO_GBK[18858] := 16#7008;
   // UNICODE_TO_GBK[18859] := 16#9E60;
   // UNICODE_TO_GBK[18860] := 16#7009;
   // UNICODE_TO_GBK[18861] := 16#9E61;
   // UNICODE_TO_GBK[18862] := 16#700A;
   // UNICODE_TO_GBK[18863] := 16#9E62;
   // UNICODE_TO_GBK[18864] := 16#700B;
   // UNICODE_TO_GBK[18865] := 16#9E63;
   // UNICODE_TO_GBK[18866] := 16#700C;
   // UNICODE_TO_GBK[18867] := 16#9E64;
   // UNICODE_TO_GBK[18868] := 16#700D;
   // UNICODE_TO_GBK[18869] := 16#9E65;
   // UNICODE_TO_GBK[18870] := 16#700E;
   // UNICODE_TO_GBK[18871] := 16#9E66;
   // UNICODE_TO_GBK[18872] := 16#700F;
   // UNICODE_TO_GBK[18873] := 16#9E67;
   // UNICODE_TO_GBK[18874] := 16#7010;
   // UNICODE_TO_GBK[18875] := 16#9E68;
   // UNICODE_TO_GBK[18876] := 16#7011;
   // UNICODE_TO_GBK[18877] := 16#C6D9;
   // UNICODE_TO_GBK[18878] := 16#7012;
   // UNICODE_TO_GBK[18879] := 16#9E69;
   // UNICODE_TO_GBK[18880] := 16#7013;
   // UNICODE_TO_GBK[18881] := 16#9E6A;
   // UNICODE_TO_GBK[18882] := 16#7014;
   // UNICODE_TO_GBK[18883] := 16#9E6B;
   // UNICODE_TO_GBK[18884] := 16#7015;
   // UNICODE_TO_GBK[18885] := 16#9E6C;
   // UNICODE_TO_GBK[18886] := 16#7016;
   // UNICODE_TO_GBK[18887] := 16#9E6D;
   // UNICODE_TO_GBK[18888] := 16#7017;
   // UNICODE_TO_GBK[18889] := 16#9E6E;
   // UNICODE_TO_GBK[18890] := 16#7018;
   // UNICODE_TO_GBK[18891] := 16#9E6F;
   // UNICODE_TO_GBK[18892] := 16#7019;
   // UNICODE_TO_GBK[18893] := 16#9E70;
   // UNICODE_TO_GBK[18894] := 16#701A;
   // UNICODE_TO_GBK[18895] := 16#E5AB;
   // UNICODE_TO_GBK[18896] := 16#701B;
   // UNICODE_TO_GBK[18897] := 16#E5AD;
   // UNICODE_TO_GBK[18898] := 16#701C;
   // UNICODE_TO_GBK[18899] := 16#9E71;
   // UNICODE_TO_GBK[18900] := 16#701D;
   // UNICODE_TO_GBK[18901] := 16#9E72;
   // UNICODE_TO_GBK[18902] := 16#701E;
   // UNICODE_TO_GBK[18903] := 16#9E73;
   // UNICODE_TO_GBK[18904] := 16#701F;
   // UNICODE_TO_GBK[18905] := 16#9E74;
   // UNICODE_TO_GBK[18906] := 16#7020;
   // UNICODE_TO_GBK[18907] := 16#9E75;
   // UNICODE_TO_GBK[18908] := 16#7021;
   // UNICODE_TO_GBK[18909] := 16#9E76;
   // UNICODE_TO_GBK[18910] := 16#7022;
   // UNICODE_TO_GBK[18911] := 16#9E77;
   // UNICODE_TO_GBK[18912] := 16#7023;
   // UNICODE_TO_GBK[18913] := 16#E5AC;
   // UNICODE_TO_GBK[18914] := 16#7024;
   // UNICODE_TO_GBK[18915] := 16#9E78;
   // UNICODE_TO_GBK[18916] := 16#7025;
   // UNICODE_TO_GBK[18917] := 16#9E79;
   // UNICODE_TO_GBK[18918] := 16#7026;
   // UNICODE_TO_GBK[18919] := 16#9E7A;
   // UNICODE_TO_GBK[18920] := 16#7027;
   // UNICODE_TO_GBK[18921] := 16#9E7B;
   // UNICODE_TO_GBK[18922] := 16#7028;
   // UNICODE_TO_GBK[18923] := 16#9E7C;
   // UNICODE_TO_GBK[18924] := 16#7029;
   // UNICODE_TO_GBK[18925] := 16#9E7D;
   // UNICODE_TO_GBK[18926] := 16#702A;
   // UNICODE_TO_GBK[18927] := 16#9E7E;
   // UNICODE_TO_GBK[18928] := 16#702B;
   // UNICODE_TO_GBK[18929] := 16#9E80;
   // UNICODE_TO_GBK[18930] := 16#702C;
   // UNICODE_TO_GBK[18931] := 16#9E81;
   // UNICODE_TO_GBK[18932] := 16#702D;
   // UNICODE_TO_GBK[18933] := 16#9E82;
   // UNICODE_TO_GBK[18934] := 16#702E;
   // UNICODE_TO_GBK[18935] := 16#9E83;
   // UNICODE_TO_GBK[18936] := 16#702F;
   // UNICODE_TO_GBK[18937] := 16#9E84;
   // UNICODE_TO_GBK[18938] := 16#7030;
   // UNICODE_TO_GBK[18939] := 16#9E85;
   // UNICODE_TO_GBK[18940] := 16#7031;
   // UNICODE_TO_GBK[18941] := 16#9E86;
   // UNICODE_TO_GBK[18942] := 16#7032;
   // UNICODE_TO_GBK[18943] := 16#9E87;
   // UNICODE_TO_GBK[18944] := 16#7033;
   // UNICODE_TO_GBK[18945] := 16#9E88;
   // UNICODE_TO_GBK[18946] := 16#7034;
   // UNICODE_TO_GBK[18947] := 16#9E89;
   // UNICODE_TO_GBK[18948] := 16#7035;
   // UNICODE_TO_GBK[18949] := 16#E5AF;
   // UNICODE_TO_GBK[18950] := 16#7036;
   // UNICODE_TO_GBK[18951] := 16#9E8A;
   // UNICODE_TO_GBK[18952] := 16#7037;
   // UNICODE_TO_GBK[18953] := 16#9E8B;
   // UNICODE_TO_GBK[18954] := 16#7038;
   // UNICODE_TO_GBK[18955] := 16#9E8C;
   // UNICODE_TO_GBK[18956] := 16#7039;
   // UNICODE_TO_GBK[18957] := 16#E5AE;
   // UNICODE_TO_GBK[18958] := 16#703A;
   // UNICODE_TO_GBK[18959] := 16#9E8D;
   // UNICODE_TO_GBK[18960] := 16#703B;
   // UNICODE_TO_GBK[18961] := 16#9E8E;
   // UNICODE_TO_GBK[18962] := 16#703C;
   // UNICODE_TO_GBK[18963] := 16#9E8F;
   // UNICODE_TO_GBK[18964] := 16#703D;
   // UNICODE_TO_GBK[18965] := 16#9E90;
   // UNICODE_TO_GBK[18966] := 16#703E;
   // UNICODE_TO_GBK[18967] := 16#9E91;
   // UNICODE_TO_GBK[18968] := 16#703F;
   // UNICODE_TO_GBK[18969] := 16#9E92;
   // UNICODE_TO_GBK[18970] := 16#7040;
   // UNICODE_TO_GBK[18971] := 16#9E93;
   // UNICODE_TO_GBK[18972] := 16#7041;
   // UNICODE_TO_GBK[18973] := 16#9E94;
   // UNICODE_TO_GBK[18974] := 16#7042;
   // UNICODE_TO_GBK[18975] := 16#9E95;
   // UNICODE_TO_GBK[18976] := 16#7043;
   // UNICODE_TO_GBK[18977] := 16#9E96;
   // UNICODE_TO_GBK[18978] := 16#7044;
   // UNICODE_TO_GBK[18979] := 16#9E97;
   // UNICODE_TO_GBK[18980] := 16#7045;
   // UNICODE_TO_GBK[18981] := 16#9E98;
   // UNICODE_TO_GBK[18982] := 16#7046;
   // UNICODE_TO_GBK[18983] := 16#9E99;
   // UNICODE_TO_GBK[18984] := 16#7047;
   // UNICODE_TO_GBK[18985] := 16#9E9A;
   // UNICODE_TO_GBK[18986] := 16#7048;
   // UNICODE_TO_GBK[18987] := 16#9E9B;
   // UNICODE_TO_GBK[18988] := 16#7049;
   // UNICODE_TO_GBK[18989] := 16#9E9C;
   // UNICODE_TO_GBK[18990] := 16#704A;
   // UNICODE_TO_GBK[18991] := 16#9E9D;
   // UNICODE_TO_GBK[18992] := 16#704B;
   // UNICODE_TO_GBK[18993] := 16#9E9E;
   // UNICODE_TO_GBK[18994] := 16#704C;
   // UNICODE_TO_GBK[18995] := 16#B9E0;
   // UNICODE_TO_GBK[18996] := 16#704D;
   // UNICODE_TO_GBK[18997] := 16#9E9F;
   // UNICODE_TO_GBK[18998] := 16#704E;
   // UNICODE_TO_GBK[18999] := 16#9EA0;
   // UNICODE_TO_GBK[19000] := 16#704F;
   // UNICODE_TO_GBK[19001] := 16#E5B0;
   // UNICODE_TO_GBK[19002] := 16#7050;
   // UNICODE_TO_GBK[19003] := 16#9EA1;
   // UNICODE_TO_GBK[19004] := 16#7051;
   // UNICODE_TO_GBK[19005] := 16#9EA2;
   // UNICODE_TO_GBK[19006] := 16#7052;
   // UNICODE_TO_GBK[19007] := 16#9EA3;
   // UNICODE_TO_GBK[19008] := 16#7053;
   // UNICODE_TO_GBK[19009] := 16#9EA4;
   // UNICODE_TO_GBK[19010] := 16#7054;
   // UNICODE_TO_GBK[19011] := 16#9EA5;
   // UNICODE_TO_GBK[19012] := 16#7055;
   // UNICODE_TO_GBK[19013] := 16#9EA6;
   // UNICODE_TO_GBK[19014] := 16#7056;
   // UNICODE_TO_GBK[19015] := 16#9EA7;
   // UNICODE_TO_GBK[19016] := 16#7057;
   // UNICODE_TO_GBK[19017] := 16#9EA8;
   // UNICODE_TO_GBK[19018] := 16#7058;
   // UNICODE_TO_GBK[19019] := 16#9EA9;
   // UNICODE_TO_GBK[19020] := 16#7059;
   // UNICODE_TO_GBK[19021] := 16#9EAA;
   // UNICODE_TO_GBK[19022] := 16#705A;
   // UNICODE_TO_GBK[19023] := 16#9EAB;
   // UNICODE_TO_GBK[19024] := 16#705B;
   // UNICODE_TO_GBK[19025] := 16#9EAC;
   // UNICODE_TO_GBK[19026] := 16#705C;
   // UNICODE_TO_GBK[19027] := 16#9EAD;
   // UNICODE_TO_GBK[19028] := 16#705D;
   // UNICODE_TO_GBK[19029] := 16#9EAE;
   // UNICODE_TO_GBK[19030] := 16#705E;
   // UNICODE_TO_GBK[19031] := 16#E5B1;
   // UNICODE_TO_GBK[19032] := 16#705F;
   // UNICODE_TO_GBK[19033] := 16#9EAF;
   // UNICODE_TO_GBK[19034] := 16#7060;
   // UNICODE_TO_GBK[19035] := 16#9EB0;
   // UNICODE_TO_GBK[19036] := 16#7061;
   // UNICODE_TO_GBK[19037] := 16#9EB1;
   // UNICODE_TO_GBK[19038] := 16#7062;
   // UNICODE_TO_GBK[19039] := 16#9EB2;
   // UNICODE_TO_GBK[19040] := 16#7063;
   // UNICODE_TO_GBK[19041] := 16#9EB3;
   // UNICODE_TO_GBK[19042] := 16#7064;
   // UNICODE_TO_GBK[19043] := 16#9EB4;
   // UNICODE_TO_GBK[19044] := 16#7065;
   // UNICODE_TO_GBK[19045] := 16#9EB5;
   // UNICODE_TO_GBK[19046] := 16#7066;
   // UNICODE_TO_GBK[19047] := 16#9EB6;
   // UNICODE_TO_GBK[19048] := 16#7067;
   // UNICODE_TO_GBK[19049] := 16#9EB7;
   // UNICODE_TO_GBK[19050] := 16#7068;
   // UNICODE_TO_GBK[19051] := 16#9EB8;
   // UNICODE_TO_GBK[19052] := 16#7069;
   // UNICODE_TO_GBK[19053] := 16#9EB9;
   // UNICODE_TO_GBK[19054] := 16#706A;
   // UNICODE_TO_GBK[19055] := 16#9EBA;
   // UNICODE_TO_GBK[19056] := 16#706B;
   // UNICODE_TO_GBK[19057] := 16#BBF0;
   // UNICODE_TO_GBK[19058] := 16#706C;
   // UNICODE_TO_GBK[19059] := 16#ECE1;
   // UNICODE_TO_GBK[19060] := 16#706D;
   // UNICODE_TO_GBK[19061] := 16#C3F0;
   // UNICODE_TO_GBK[19062] := 16#706E;
   // UNICODE_TO_GBK[19063] := 16#9EBB;
   // UNICODE_TO_GBK[19064] := 16#706F;
   // UNICODE_TO_GBK[19065] := 16#B5C6;
   // UNICODE_TO_GBK[19066] := 16#7070;
   // UNICODE_TO_GBK[19067] := 16#BBD2;
   // UNICODE_TO_GBK[19068] := 16#7071;
   // UNICODE_TO_GBK[19069] := 16#9EBC;
   // UNICODE_TO_GBK[19070] := 16#7072;
   // UNICODE_TO_GBK[19071] := 16#9EBD;
   // UNICODE_TO_GBK[19072] := 16#7073;
   // UNICODE_TO_GBK[19073] := 16#9EBE;
   // UNICODE_TO_GBK[19074] := 16#7074;
   // UNICODE_TO_GBK[19075] := 16#9EBF;
   // UNICODE_TO_GBK[19076] := 16#7075;
   // UNICODE_TO_GBK[19077] := 16#C1E9;
   // UNICODE_TO_GBK[19078] := 16#7076;
   // UNICODE_TO_GBK[19079] := 16#D4EE;
   // UNICODE_TO_GBK[19080] := 16#7077;
   // UNICODE_TO_GBK[19081] := 16#9EC0;
   // UNICODE_TO_GBK[19082] := 16#7078;
   // UNICODE_TO_GBK[19083] := 16#BEC4;
   // UNICODE_TO_GBK[19084] := 16#7079;
   // UNICODE_TO_GBK[19085] := 16#9EC1;
   // UNICODE_TO_GBK[19086] := 16#707A;
   // UNICODE_TO_GBK[19087] := 16#9EC2;
   // UNICODE_TO_GBK[19088] := 16#707B;
   // UNICODE_TO_GBK[19089] := 16#9EC3;
   // UNICODE_TO_GBK[19090] := 16#707C;
   // UNICODE_TO_GBK[19091] := 16#D7C6;
   // UNICODE_TO_GBK[19092] := 16#707D;
   // UNICODE_TO_GBK[19093] := 16#9EC4;
   // UNICODE_TO_GBK[19094] := 16#707E;
   // UNICODE_TO_GBK[19095] := 16#D4D6;
   // UNICODE_TO_GBK[19096] := 16#707F;
   // UNICODE_TO_GBK[19097] := 16#B2D3;
   // UNICODE_TO_GBK[19098] := 16#7080;
   // UNICODE_TO_GBK[19099] := 16#ECBE;
   // UNICODE_TO_GBK[19100] := 16#7081;
   // UNICODE_TO_GBK[19101] := 16#9EC5;
   // UNICODE_TO_GBK[19102] := 16#7082;
   // UNICODE_TO_GBK[19103] := 16#9EC6;
   // UNICODE_TO_GBK[19104] := 16#7083;
   // UNICODE_TO_GBK[19105] := 16#9EC7;
   // UNICODE_TO_GBK[19106] := 16#7084;
   // UNICODE_TO_GBK[19107] := 16#9EC8;
   // UNICODE_TO_GBK[19108] := 16#7085;
   // UNICODE_TO_GBK[19109] := 16#EAC1;
   // UNICODE_TO_GBK[19110] := 16#7086;
   // UNICODE_TO_GBK[19111] := 16#9EC9;
   // UNICODE_TO_GBK[19112] := 16#7087;
   // UNICODE_TO_GBK[19113] := 16#9ECA;
   // UNICODE_TO_GBK[19114] := 16#7088;
   // UNICODE_TO_GBK[19115] := 16#9ECB;
   // UNICODE_TO_GBK[19116] := 16#7089;
   // UNICODE_TO_GBK[19117] := 16#C2AF;
   // UNICODE_TO_GBK[19118] := 16#708A;
   // UNICODE_TO_GBK[19119] := 16#B4B6;
   // UNICODE_TO_GBK[19120] := 16#708B;
   // UNICODE_TO_GBK[19121] := 16#9ECC;
   // UNICODE_TO_GBK[19122] := 16#708C;
   // UNICODE_TO_GBK[19123] := 16#9ECD;
   // UNICODE_TO_GBK[19124] := 16#708D;
   // UNICODE_TO_GBK[19125] := 16#9ECE;
   // UNICODE_TO_GBK[19126] := 16#708E;
   // UNICODE_TO_GBK[19127] := 16#D1D7;
   // UNICODE_TO_GBK[19128] := 16#708F;
   // UNICODE_TO_GBK[19129] := 16#9ECF;
   // UNICODE_TO_GBK[19130] := 16#7090;
   // UNICODE_TO_GBK[19131] := 16#9ED0;
   // UNICODE_TO_GBK[19132] := 16#7091;
   // UNICODE_TO_GBK[19133] := 16#9ED1;
   // UNICODE_TO_GBK[19134] := 16#7092;
   // UNICODE_TO_GBK[19135] := 16#B3B4;
   // UNICODE_TO_GBK[19136] := 16#7093;
   // UNICODE_TO_GBK[19137] := 16#9ED2;
   // UNICODE_TO_GBK[19138] := 16#7094;
   // UNICODE_TO_GBK[19139] := 16#C8B2;
   // UNICODE_TO_GBK[19140] := 16#7095;
   // UNICODE_TO_GBK[19141] := 16#BFBB;
   // UNICODE_TO_GBK[19142] := 16#7096;
   // UNICODE_TO_GBK[19143] := 16#ECC0;
   // UNICODE_TO_GBK[19144] := 16#7097;
   // UNICODE_TO_GBK[19145] := 16#9ED3;
   // UNICODE_TO_GBK[19146] := 16#7098;
   // UNICODE_TO_GBK[19147] := 16#9ED4;
   // UNICODE_TO_GBK[19148] := 16#7099;
   // UNICODE_TO_GBK[19149] := 16#D6CB;
   // UNICODE_TO_GBK[19150] := 16#709A;
   // UNICODE_TO_GBK[19151] := 16#9ED5;
   // UNICODE_TO_GBK[19152] := 16#709B;
   // UNICODE_TO_GBK[19153] := 16#9ED6;
   // UNICODE_TO_GBK[19154] := 16#709C;
   // UNICODE_TO_GBK[19155] := 16#ECBF;
   // UNICODE_TO_GBK[19156] := 16#709D;
   // UNICODE_TO_GBK[19157] := 16#ECC1;
   // UNICODE_TO_GBK[19158] := 16#709E;
   // UNICODE_TO_GBK[19159] := 16#9ED7;
   // UNICODE_TO_GBK[19160] := 16#709F;
   // UNICODE_TO_GBK[19161] := 16#9ED8;
   // UNICODE_TO_GBK[19162] := 16#70A0;
   // UNICODE_TO_GBK[19163] := 16#9ED9;
   // UNICODE_TO_GBK[19164] := 16#70A1;
   // UNICODE_TO_GBK[19165] := 16#9EDA;
   // UNICODE_TO_GBK[19166] := 16#70A2;
   // UNICODE_TO_GBK[19167] := 16#9EDB;
   // UNICODE_TO_GBK[19168] := 16#70A3;
   // UNICODE_TO_GBK[19169] := 16#9EDC;
   // UNICODE_TO_GBK[19170] := 16#70A4;
   // UNICODE_TO_GBK[19171] := 16#9EDD;
   // UNICODE_TO_GBK[19172] := 16#70A5;
   // UNICODE_TO_GBK[19173] := 16#9EDE;
   // UNICODE_TO_GBK[19174] := 16#70A6;
   // UNICODE_TO_GBK[19175] := 16#9EDF;
   // UNICODE_TO_GBK[19176] := 16#70A7;
   // UNICODE_TO_GBK[19177] := 16#9EE0;
   // UNICODE_TO_GBK[19178] := 16#70A8;
   // UNICODE_TO_GBK[19179] := 16#9EE1;
   // UNICODE_TO_GBK[19180] := 16#70A9;
   // UNICODE_TO_GBK[19181] := 16#9EE2;
   // UNICODE_TO_GBK[19182] := 16#70AA;
   // UNICODE_TO_GBK[19183] := 16#9EE3;
   // UNICODE_TO_GBK[19184] := 16#70AB;
   // UNICODE_TO_GBK[19185] := 16#ECC5;
   // UNICODE_TO_GBK[19186] := 16#70AC;
   // UNICODE_TO_GBK[19187] := 16#BEE6;
   // UNICODE_TO_GBK[19188] := 16#70AD;
   // UNICODE_TO_GBK[19189] := 16#CCBF;
   // UNICODE_TO_GBK[19190] := 16#70AE;
   // UNICODE_TO_GBK[19191] := 16#C5DA;
   // UNICODE_TO_GBK[19192] := 16#70AF;
   // UNICODE_TO_GBK[19193] := 16#BEBC;
   // UNICODE_TO_GBK[19194] := 16#70B0;
   // UNICODE_TO_GBK[19195] := 16#9EE4;
   // UNICODE_TO_GBK[19196] := 16#70B1;
   // UNICODE_TO_GBK[19197] := 16#ECC6;
   // UNICODE_TO_GBK[19198] := 16#70B2;
   // UNICODE_TO_GBK[19199] := 16#9EE5;
   // UNICODE_TO_GBK[19200] := 16#70B3;
   // UNICODE_TO_GBK[19201] := 16#B1FE;
   // UNICODE_TO_GBK[19202] := 16#70B4;
   // UNICODE_TO_GBK[19203] := 16#9EE6;
   // UNICODE_TO_GBK[19204] := 16#70B5;
   // UNICODE_TO_GBK[19205] := 16#9EE7;
   // UNICODE_TO_GBK[19206] := 16#70B6;
   // UNICODE_TO_GBK[19207] := 16#9EE8;
   // UNICODE_TO_GBK[19208] := 16#70B7;
   // UNICODE_TO_GBK[19209] := 16#ECC4;
   // UNICODE_TO_GBK[19210] := 16#70B8;
   // UNICODE_TO_GBK[19211] := 16#D5A8;
   // UNICODE_TO_GBK[19212] := 16#70B9;
   // UNICODE_TO_GBK[19213] := 16#B5E3;
   // UNICODE_TO_GBK[19214] := 16#70BA;
   // UNICODE_TO_GBK[19215] := 16#9EE9;
   // UNICODE_TO_GBK[19216] := 16#70BB;
   // UNICODE_TO_GBK[19217] := 16#ECC2;
   // UNICODE_TO_GBK[19218] := 16#70BC;
   // UNICODE_TO_GBK[19219] := 16#C1B6;
   // UNICODE_TO_GBK[19220] := 16#70BD;
   // UNICODE_TO_GBK[19221] := 16#B3E3;
   // UNICODE_TO_GBK[19222] := 16#70BE;
   // UNICODE_TO_GBK[19223] := 16#9EEA;
   // UNICODE_TO_GBK[19224] := 16#70BF;
   // UNICODE_TO_GBK[19225] := 16#9EEB;
   // UNICODE_TO_GBK[19226] := 16#70C0;
   // UNICODE_TO_GBK[19227] := 16#ECC3;
   // UNICODE_TO_GBK[19228] := 16#70C1;
   // UNICODE_TO_GBK[19229] := 16#CBB8;
   // UNICODE_TO_GBK[19230] := 16#70C2;
   // UNICODE_TO_GBK[19231] := 16#C0C3;
   // UNICODE_TO_GBK[19232] := 16#70C3;
   // UNICODE_TO_GBK[19233] := 16#CCFE;
   // UNICODE_TO_GBK[19234] := 16#70C4;
   // UNICODE_TO_GBK[19235] := 16#9EEC;
   // UNICODE_TO_GBK[19236] := 16#70C5;
   // UNICODE_TO_GBK[19237] := 16#9EED;
   // UNICODE_TO_GBK[19238] := 16#70C6;
   // UNICODE_TO_GBK[19239] := 16#9EEE;
   // UNICODE_TO_GBK[19240] := 16#70C7;
   // UNICODE_TO_GBK[19241] := 16#9EEF;
   // UNICODE_TO_GBK[19242] := 16#70C8;
   // UNICODE_TO_GBK[19243] := 16#C1D2;
   // UNICODE_TO_GBK[19244] := 16#70C9;
   // UNICODE_TO_GBK[19245] := 16#9EF0;
   // UNICODE_TO_GBK[19246] := 16#70CA;
   // UNICODE_TO_GBK[19247] := 16#ECC8;
   // UNICODE_TO_GBK[19248] := 16#70CB;
   // UNICODE_TO_GBK[19249] := 16#9EF1;
   // UNICODE_TO_GBK[19250] := 16#70CC;
   // UNICODE_TO_GBK[19251] := 16#9EF2;
   // UNICODE_TO_GBK[19252] := 16#70CD;
   // UNICODE_TO_GBK[19253] := 16#9EF3;
   // UNICODE_TO_GBK[19254] := 16#70CE;
   // UNICODE_TO_GBK[19255] := 16#9EF4;
   // UNICODE_TO_GBK[19256] := 16#70CF;
   // UNICODE_TO_GBK[19257] := 16#9EF5;
   // UNICODE_TO_GBK[19258] := 16#70D0;
   // UNICODE_TO_GBK[19259] := 16#9EF6;
   // UNICODE_TO_GBK[19260] := 16#70D1;
   // UNICODE_TO_GBK[19261] := 16#9EF7;
   // UNICODE_TO_GBK[19262] := 16#70D2;
   // UNICODE_TO_GBK[19263] := 16#9EF8;
   // UNICODE_TO_GBK[19264] := 16#70D3;
   // UNICODE_TO_GBK[19265] := 16#9EF9;
   // UNICODE_TO_GBK[19266] := 16#70D4;
   // UNICODE_TO_GBK[19267] := 16#9EFA;
   // UNICODE_TO_GBK[19268] := 16#70D5;
   // UNICODE_TO_GBK[19269] := 16#9EFB;
   // UNICODE_TO_GBK[19270] := 16#70D6;
   // UNICODE_TO_GBK[19271] := 16#9EFC;
   // UNICODE_TO_GBK[19272] := 16#70D7;
   // UNICODE_TO_GBK[19273] := 16#9EFD;
   // UNICODE_TO_GBK[19274] := 16#70D8;
   // UNICODE_TO_GBK[19275] := 16#BAE6;
   // UNICODE_TO_GBK[19276] := 16#70D9;
   // UNICODE_TO_GBK[19277] := 16#C0D3;
   // UNICODE_TO_GBK[19278] := 16#70DA;
   // UNICODE_TO_GBK[19279] := 16#9EFE;
   // UNICODE_TO_GBK[19280] := 16#70DB;
   // UNICODE_TO_GBK[19281] := 16#D6F2;
   // UNICODE_TO_GBK[19282] := 16#70DC;
   // UNICODE_TO_GBK[19283] := 16#9F40;
   // UNICODE_TO_GBK[19284] := 16#70DD;
   // UNICODE_TO_GBK[19285] := 16#9F41;
   // UNICODE_TO_GBK[19286] := 16#70DE;
   // UNICODE_TO_GBK[19287] := 16#9F42;
   // UNICODE_TO_GBK[19288] := 16#70DF;
   // UNICODE_TO_GBK[19289] := 16#D1CC;
   // UNICODE_TO_GBK[19290] := 16#70E0;
   // UNICODE_TO_GBK[19291] := 16#9F43;
   // UNICODE_TO_GBK[19292] := 16#70E1;
   // UNICODE_TO_GBK[19293] := 16#9F44;
   // UNICODE_TO_GBK[19294] := 16#70E2;
   // UNICODE_TO_GBK[19295] := 16#9F45;
   // UNICODE_TO_GBK[19296] := 16#70E3;
   // UNICODE_TO_GBK[19297] := 16#9F46;
   // UNICODE_TO_GBK[19298] := 16#70E4;
   // UNICODE_TO_GBK[19299] := 16#BFBE;
   // UNICODE_TO_GBK[19300] := 16#70E5;
   // UNICODE_TO_GBK[19301] := 16#9F47;
   // UNICODE_TO_GBK[19302] := 16#70E6;
   // UNICODE_TO_GBK[19303] := 16#B7B3;
   // UNICODE_TO_GBK[19304] := 16#70E7;
   // UNICODE_TO_GBK[19305] := 16#C9D5;
   // UNICODE_TO_GBK[19306] := 16#70E8;
   // UNICODE_TO_GBK[19307] := 16#ECC7;
   // UNICODE_TO_GBK[19308] := 16#70E9;
   // UNICODE_TO_GBK[19309] := 16#BBE2;
   // UNICODE_TO_GBK[19310] := 16#70EA;
   // UNICODE_TO_GBK[19311] := 16#9F48;
   // UNICODE_TO_GBK[19312] := 16#70EB;
   // UNICODE_TO_GBK[19313] := 16#CCCC;
   // UNICODE_TO_GBK[19314] := 16#70EC;
   // UNICODE_TO_GBK[19315] := 16#BDFD;
   // UNICODE_TO_GBK[19316] := 16#70ED;
   // UNICODE_TO_GBK[19317] := 16#C8C8;
   // UNICODE_TO_GBK[19318] := 16#70EE;
   // UNICODE_TO_GBK[19319] := 16#9F49;
   // UNICODE_TO_GBK[19320] := 16#70EF;
   // UNICODE_TO_GBK[19321] := 16#CFA9;
   // UNICODE_TO_GBK[19322] := 16#70F0;
   // UNICODE_TO_GBK[19323] := 16#9F4A;
   // UNICODE_TO_GBK[19324] := 16#70F1;
   // UNICODE_TO_GBK[19325] := 16#9F4B;
   // UNICODE_TO_GBK[19326] := 16#70F2;
   // UNICODE_TO_GBK[19327] := 16#9F4C;
   // UNICODE_TO_GBK[19328] := 16#70F3;
   // UNICODE_TO_GBK[19329] := 16#9F4D;
   // UNICODE_TO_GBK[19330] := 16#70F4;
   // UNICODE_TO_GBK[19331] := 16#9F4E;
   // UNICODE_TO_GBK[19332] := 16#70F5;
   // UNICODE_TO_GBK[19333] := 16#9F4F;
   // UNICODE_TO_GBK[19334] := 16#70F6;
   // UNICODE_TO_GBK[19335] := 16#9F50;
   // UNICODE_TO_GBK[19336] := 16#70F7;
   // UNICODE_TO_GBK[19337] := 16#CDE9;
   // UNICODE_TO_GBK[19338] := 16#70F8;
   // UNICODE_TO_GBK[19339] := 16#9F51;
   // UNICODE_TO_GBK[19340] := 16#70F9;
   // UNICODE_TO_GBK[19341] := 16#C5EB;
   // UNICODE_TO_GBK[19342] := 16#70FA;
   // UNICODE_TO_GBK[19343] := 16#9F52;
   // UNICODE_TO_GBK[19344] := 16#70FB;
   // UNICODE_TO_GBK[19345] := 16#9F53;
   // UNICODE_TO_GBK[19346] := 16#70FC;
   // UNICODE_TO_GBK[19347] := 16#9F54;
   // UNICODE_TO_GBK[19348] := 16#70FD;
   // UNICODE_TO_GBK[19349] := 16#B7E9;
   // UNICODE_TO_GBK[19350] := 16#70FE;
   // UNICODE_TO_GBK[19351] := 16#9F55;
   // UNICODE_TO_GBK[19352] := 16#70FF;
   // UNICODE_TO_GBK[19353] := 16#9F56;
   // UNICODE_TO_GBK[19354] := 16#7100;
   // UNICODE_TO_GBK[19355] := 16#9F57;
   // UNICODE_TO_GBK[19356] := 16#7101;
   // UNICODE_TO_GBK[19357] := 16#9F58;
   // UNICODE_TO_GBK[19358] := 16#7102;
   // UNICODE_TO_GBK[19359] := 16#9F59;
   // UNICODE_TO_GBK[19360] := 16#7103;
   // UNICODE_TO_GBK[19361] := 16#9F5A;
   // UNICODE_TO_GBK[19362] := 16#7104;
   // UNICODE_TO_GBK[19363] := 16#9F5B;
   // UNICODE_TO_GBK[19364] := 16#7105;
   // UNICODE_TO_GBK[19365] := 16#9F5C;
   // UNICODE_TO_GBK[19366] := 16#7106;
   // UNICODE_TO_GBK[19367] := 16#9F5D;
   // UNICODE_TO_GBK[19368] := 16#7107;
   // UNICODE_TO_GBK[19369] := 16#9F5E;
   // UNICODE_TO_GBK[19370] := 16#7108;
   // UNICODE_TO_GBK[19371] := 16#9F5F;
   // UNICODE_TO_GBK[19372] := 16#7109;
   // UNICODE_TO_GBK[19373] := 16#D1C9;
   // UNICODE_TO_GBK[19374] := 16#710A;
   // UNICODE_TO_GBK[19375] := 16#BAB8;
   // UNICODE_TO_GBK[19376] := 16#710B;
   // UNICODE_TO_GBK[19377] := 16#9F60;
   // UNICODE_TO_GBK[19378] := 16#710C;
   // UNICODE_TO_GBK[19379] := 16#9F61;
   // UNICODE_TO_GBK[19380] := 16#710D;
   // UNICODE_TO_GBK[19381] := 16#9F62;
   // UNICODE_TO_GBK[19382] := 16#710E;
   // UNICODE_TO_GBK[19383] := 16#9F63;
   // UNICODE_TO_GBK[19384] := 16#710F;
   // UNICODE_TO_GBK[19385] := 16#9F64;
   // UNICODE_TO_GBK[19386] := 16#7110;
   // UNICODE_TO_GBK[19387] := 16#ECC9;
   // UNICODE_TO_GBK[19388] := 16#7111;
   // UNICODE_TO_GBK[19389] := 16#9F65;
   // UNICODE_TO_GBK[19390] := 16#7112;
   // UNICODE_TO_GBK[19391] := 16#9F66;
   // UNICODE_TO_GBK[19392] := 16#7113;
   // UNICODE_TO_GBK[19393] := 16#ECCA;
   // UNICODE_TO_GBK[19394] := 16#7114;
   // UNICODE_TO_GBK[19395] := 16#9F67;
   // UNICODE_TO_GBK[19396] := 16#7115;
   // UNICODE_TO_GBK[19397] := 16#BBC0;
   // UNICODE_TO_GBK[19398] := 16#7116;
   // UNICODE_TO_GBK[19399] := 16#ECCB;
   // UNICODE_TO_GBK[19400] := 16#7117;
   // UNICODE_TO_GBK[19401] := 16#9F68;
   // UNICODE_TO_GBK[19402] := 16#7118;
   // UNICODE_TO_GBK[19403] := 16#ECE2;
   // UNICODE_TO_GBK[19404] := 16#7119;
   // UNICODE_TO_GBK[19405] := 16#B1BA;
   // UNICODE_TO_GBK[19406] := 16#711A;
   // UNICODE_TO_GBK[19407] := 16#B7D9;
   // UNICODE_TO_GBK[19408] := 16#711B;
   // UNICODE_TO_GBK[19409] := 16#9F69;
   // UNICODE_TO_GBK[19410] := 16#711C;
   // UNICODE_TO_GBK[19411] := 16#9F6A;
   // UNICODE_TO_GBK[19412] := 16#711D;
   // UNICODE_TO_GBK[19413] := 16#9F6B;
   // UNICODE_TO_GBK[19414] := 16#711E;
   // UNICODE_TO_GBK[19415] := 16#9F6C;
   // UNICODE_TO_GBK[19416] := 16#711F;
   // UNICODE_TO_GBK[19417] := 16#9F6D;
   // UNICODE_TO_GBK[19418] := 16#7120;
   // UNICODE_TO_GBK[19419] := 16#9F6E;
   // UNICODE_TO_GBK[19420] := 16#7121;
   // UNICODE_TO_GBK[19421] := 16#9F6F;
   // UNICODE_TO_GBK[19422] := 16#7122;
   // UNICODE_TO_GBK[19423] := 16#9F70;
   // UNICODE_TO_GBK[19424] := 16#7123;
   // UNICODE_TO_GBK[19425] := 16#9F71;
   // UNICODE_TO_GBK[19426] := 16#7124;
   // UNICODE_TO_GBK[19427] := 16#9F72;
   // UNICODE_TO_GBK[19428] := 16#7125;
   // UNICODE_TO_GBK[19429] := 16#9F73;
   // UNICODE_TO_GBK[19430] := 16#7126;
   // UNICODE_TO_GBK[19431] := 16#BDB9;
   // UNICODE_TO_GBK[19432] := 16#7127;
   // UNICODE_TO_GBK[19433] := 16#9F74;
   // UNICODE_TO_GBK[19434] := 16#7128;
   // UNICODE_TO_GBK[19435] := 16#9F75;
   // UNICODE_TO_GBK[19436] := 16#7129;
   // UNICODE_TO_GBK[19437] := 16#9F76;
   // UNICODE_TO_GBK[19438] := 16#712A;
   // UNICODE_TO_GBK[19439] := 16#9F77;
   // UNICODE_TO_GBK[19440] := 16#712B;
   // UNICODE_TO_GBK[19441] := 16#9F78;
   // UNICODE_TO_GBK[19442] := 16#712C;
   // UNICODE_TO_GBK[19443] := 16#9F79;
   // UNICODE_TO_GBK[19444] := 16#712D;
   // UNICODE_TO_GBK[19445] := 16#9F7A;
   // UNICODE_TO_GBK[19446] := 16#712E;
   // UNICODE_TO_GBK[19447] := 16#9F7B;
   // UNICODE_TO_GBK[19448] := 16#712F;
   // UNICODE_TO_GBK[19449] := 16#ECCC;
   // UNICODE_TO_GBK[19450] := 16#7130;
   // UNICODE_TO_GBK[19451] := 16#D1E6;
   // UNICODE_TO_GBK[19452] := 16#7131;
   // UNICODE_TO_GBK[19453] := 16#ECCD;
   // UNICODE_TO_GBK[19454] := 16#7132;
   // UNICODE_TO_GBK[19455] := 16#9F7C;
   // UNICODE_TO_GBK[19456] := 16#7133;
   // UNICODE_TO_GBK[19457] := 16#9F7D;
   // UNICODE_TO_GBK[19458] := 16#7134;
   // UNICODE_TO_GBK[19459] := 16#9F7E;
   // UNICODE_TO_GBK[19460] := 16#7135;
   // UNICODE_TO_GBK[19461] := 16#9F80;
   // UNICODE_TO_GBK[19462] := 16#7136;
   // UNICODE_TO_GBK[19463] := 16#C8BB;
   // UNICODE_TO_GBK[19464] := 16#7137;
   // UNICODE_TO_GBK[19465] := 16#9F81;
   // UNICODE_TO_GBK[19466] := 16#7138;
   // UNICODE_TO_GBK[19467] := 16#9F82;
   // UNICODE_TO_GBK[19468] := 16#7139;
   // UNICODE_TO_GBK[19469] := 16#9F83;
   // UNICODE_TO_GBK[19470] := 16#713A;
   // UNICODE_TO_GBK[19471] := 16#9F84;
   // UNICODE_TO_GBK[19472] := 16#713B;
   // UNICODE_TO_GBK[19473] := 16#9F85;
   // UNICODE_TO_GBK[19474] := 16#713C;
   // UNICODE_TO_GBK[19475] := 16#9F86;
   // UNICODE_TO_GBK[19476] := 16#713D;
   // UNICODE_TO_GBK[19477] := 16#9F87;
   // UNICODE_TO_GBK[19478] := 16#713E;
   // UNICODE_TO_GBK[19479] := 16#9F88;
   // UNICODE_TO_GBK[19480] := 16#713F;
   // UNICODE_TO_GBK[19481] := 16#9F89;
   // UNICODE_TO_GBK[19482] := 16#7140;
   // UNICODE_TO_GBK[19483] := 16#9F8A;
   // UNICODE_TO_GBK[19484] := 16#7141;
   // UNICODE_TO_GBK[19485] := 16#9F8B;
   // UNICODE_TO_GBK[19486] := 16#7142;
   // UNICODE_TO_GBK[19487] := 16#9F8C;
   // UNICODE_TO_GBK[19488] := 16#7143;
   // UNICODE_TO_GBK[19489] := 16#9F8D;
   // UNICODE_TO_GBK[19490] := 16#7144;
   // UNICODE_TO_GBK[19491] := 16#9F8E;
   // UNICODE_TO_GBK[19492] := 16#7145;
   // UNICODE_TO_GBK[19493] := 16#ECD1;
   // UNICODE_TO_GBK[19494] := 16#7146;
   // UNICODE_TO_GBK[19495] := 16#9F8F;
   // UNICODE_TO_GBK[19496] := 16#7147;
   // UNICODE_TO_GBK[19497] := 16#9F90;
   // UNICODE_TO_GBK[19498] := 16#7148;
   // UNICODE_TO_GBK[19499] := 16#9F91;
   // UNICODE_TO_GBK[19500] := 16#7149;
   // UNICODE_TO_GBK[19501] := 16#9F92;
   // UNICODE_TO_GBK[19502] := 16#714A;
   // UNICODE_TO_GBK[19503] := 16#ECD3;
   // UNICODE_TO_GBK[19504] := 16#714B;
   // UNICODE_TO_GBK[19505] := 16#9F93;
   // UNICODE_TO_GBK[19506] := 16#714C;
   // UNICODE_TO_GBK[19507] := 16#BBCD;
   // UNICODE_TO_GBK[19508] := 16#714D;
   // UNICODE_TO_GBK[19509] := 16#9F94;
   // UNICODE_TO_GBK[19510] := 16#714E;
   // UNICODE_TO_GBK[19511] := 16#BCE5;
   // UNICODE_TO_GBK[19512] := 16#714F;
   // UNICODE_TO_GBK[19513] := 16#9F95;
   // UNICODE_TO_GBK[19514] := 16#7150;
   // UNICODE_TO_GBK[19515] := 16#9F96;
   // UNICODE_TO_GBK[19516] := 16#7151;
   // UNICODE_TO_GBK[19517] := 16#9F97;
   // UNICODE_TO_GBK[19518] := 16#7152;
   // UNICODE_TO_GBK[19519] := 16#9F98;
   // UNICODE_TO_GBK[19520] := 16#7153;
   // UNICODE_TO_GBK[19521] := 16#9F99;
   // UNICODE_TO_GBK[19522] := 16#7154;
   // UNICODE_TO_GBK[19523] := 16#9F9A;
   // UNICODE_TO_GBK[19524] := 16#7155;
   // UNICODE_TO_GBK[19525] := 16#9F9B;
   // UNICODE_TO_GBK[19526] := 16#7156;
   // UNICODE_TO_GBK[19527] := 16#9F9C;
   // UNICODE_TO_GBK[19528] := 16#7157;
   // UNICODE_TO_GBK[19529] := 16#9F9D;
   // UNICODE_TO_GBK[19530] := 16#7158;
   // UNICODE_TO_GBK[19531] := 16#9F9E;
   // UNICODE_TO_GBK[19532] := 16#7159;
   // UNICODE_TO_GBK[19533] := 16#9F9F;
   // UNICODE_TO_GBK[19534] := 16#715A;
   // UNICODE_TO_GBK[19535] := 16#9FA0;
   // UNICODE_TO_GBK[19536] := 16#715B;
   // UNICODE_TO_GBK[19537] := 16#9FA1;
   // UNICODE_TO_GBK[19538] := 16#715C;
   // UNICODE_TO_GBK[19539] := 16#ECCF;
   // UNICODE_TO_GBK[19540] := 16#715D;
   // UNICODE_TO_GBK[19541] := 16#9FA2;
   // UNICODE_TO_GBK[19542] := 16#715E;
   // UNICODE_TO_GBK[19543] := 16#C9B7;
   // UNICODE_TO_GBK[19544] := 16#715F;
   // UNICODE_TO_GBK[19545] := 16#9FA3;
   // UNICODE_TO_GBK[19546] := 16#7160;
   // UNICODE_TO_GBK[19547] := 16#9FA4;
   // UNICODE_TO_GBK[19548] := 16#7161;
   // UNICODE_TO_GBK[19549] := 16#9FA5;
   // UNICODE_TO_GBK[19550] := 16#7162;
   // UNICODE_TO_GBK[19551] := 16#9FA6;
   // UNICODE_TO_GBK[19552] := 16#7163;
   // UNICODE_TO_GBK[19553] := 16#9FA7;
   // UNICODE_TO_GBK[19554] := 16#7164;
   // UNICODE_TO_GBK[19555] := 16#C3BA;
   // UNICODE_TO_GBK[19556] := 16#7165;
   // UNICODE_TO_GBK[19557] := 16#9FA8;
   // UNICODE_TO_GBK[19558] := 16#7166;
   // UNICODE_TO_GBK[19559] := 16#ECE3;
   // UNICODE_TO_GBK[19560] := 16#7167;
   // UNICODE_TO_GBK[19561] := 16#D5D5;
   // UNICODE_TO_GBK[19562] := 16#7168;
   // UNICODE_TO_GBK[19563] := 16#ECD0;
   // UNICODE_TO_GBK[19564] := 16#7169;
   // UNICODE_TO_GBK[19565] := 16#9FA9;
   // UNICODE_TO_GBK[19566] := 16#716A;
   // UNICODE_TO_GBK[19567] := 16#9FAA;
   // UNICODE_TO_GBK[19568] := 16#716B;
   // UNICODE_TO_GBK[19569] := 16#9FAB;
   // UNICODE_TO_GBK[19570] := 16#716C;
   // UNICODE_TO_GBK[19571] := 16#9FAC;
   // UNICODE_TO_GBK[19572] := 16#716D;
   // UNICODE_TO_GBK[19573] := 16#9FAD;
   // UNICODE_TO_GBK[19574] := 16#716E;
   // UNICODE_TO_GBK[19575] := 16#D6F3;
   // UNICODE_TO_GBK[19576] := 16#716F;
   // UNICODE_TO_GBK[19577] := 16#9FAE;
   // UNICODE_TO_GBK[19578] := 16#7170;
   // UNICODE_TO_GBK[19579] := 16#9FAF;
   // UNICODE_TO_GBK[19580] := 16#7171;
   // UNICODE_TO_GBK[19581] := 16#9FB0;
   // UNICODE_TO_GBK[19582] := 16#7172;
   // UNICODE_TO_GBK[19583] := 16#ECD2;
   // UNICODE_TO_GBK[19584] := 16#7173;
   // UNICODE_TO_GBK[19585] := 16#ECCE;
   // UNICODE_TO_GBK[19586] := 16#7174;
   // UNICODE_TO_GBK[19587] := 16#9FB1;
   // UNICODE_TO_GBK[19588] := 16#7175;
   // UNICODE_TO_GBK[19589] := 16#9FB2;
   // UNICODE_TO_GBK[19590] := 16#7176;
   // UNICODE_TO_GBK[19591] := 16#9FB3;
   // UNICODE_TO_GBK[19592] := 16#7177;
   // UNICODE_TO_GBK[19593] := 16#9FB4;
   // UNICODE_TO_GBK[19594] := 16#7178;
   // UNICODE_TO_GBK[19595] := 16#ECD4;
   // UNICODE_TO_GBK[19596] := 16#7179;
   // UNICODE_TO_GBK[19597] := 16#9FB5;
   // UNICODE_TO_GBK[19598] := 16#717A;
   // UNICODE_TO_GBK[19599] := 16#ECD5;
   // UNICODE_TO_GBK[19600] := 16#717B;
   // UNICODE_TO_GBK[19601] := 16#9FB6;
   // UNICODE_TO_GBK[19602] := 16#717C;
   // UNICODE_TO_GBK[19603] := 16#9FB7;
   // UNICODE_TO_GBK[19604] := 16#717D;
   // UNICODE_TO_GBK[19605] := 16#C9BF;
   // UNICODE_TO_GBK[19606] := 16#717E;
   // UNICODE_TO_GBK[19607] := 16#9FB8;
   // UNICODE_TO_GBK[19608] := 16#717F;
   // UNICODE_TO_GBK[19609] := 16#9FB9;
   // UNICODE_TO_GBK[19610] := 16#7180;
   // UNICODE_TO_GBK[19611] := 16#9FBA;
   // UNICODE_TO_GBK[19612] := 16#7181;
   // UNICODE_TO_GBK[19613] := 16#9FBB;
   // UNICODE_TO_GBK[19614] := 16#7182;
   // UNICODE_TO_GBK[19615] := 16#9FBC;
   // UNICODE_TO_GBK[19616] := 16#7183;
   // UNICODE_TO_GBK[19617] := 16#9FBD;
   // UNICODE_TO_GBK[19618] := 16#7184;
   // UNICODE_TO_GBK[19619] := 16#CFA8;
   // UNICODE_TO_GBK[19620] := 16#7185;
   // UNICODE_TO_GBK[19621] := 16#9FBE;
   // UNICODE_TO_GBK[19622] := 16#7186;
   // UNICODE_TO_GBK[19623] := 16#9FBF;
   // UNICODE_TO_GBK[19624] := 16#7187;
   // UNICODE_TO_GBK[19625] := 16#9FC0;
   // UNICODE_TO_GBK[19626] := 16#7188;
   // UNICODE_TO_GBK[19627] := 16#9FC1;
   // UNICODE_TO_GBK[19628] := 16#7189;
   // UNICODE_TO_GBK[19629] := 16#9FC2;
   // UNICODE_TO_GBK[19630] := 16#718A;
   // UNICODE_TO_GBK[19631] := 16#D0DC;
   // UNICODE_TO_GBK[19632] := 16#718B;
   // UNICODE_TO_GBK[19633] := 16#9FC3;
   // UNICODE_TO_GBK[19634] := 16#718C;
   // UNICODE_TO_GBK[19635] := 16#9FC4;
   // UNICODE_TO_GBK[19636] := 16#718D;
   // UNICODE_TO_GBK[19637] := 16#9FC5;
   // UNICODE_TO_GBK[19638] := 16#718E;
   // UNICODE_TO_GBK[19639] := 16#9FC6;
   // UNICODE_TO_GBK[19640] := 16#718F;
   // UNICODE_TO_GBK[19641] := 16#D1AC;
   // UNICODE_TO_GBK[19642] := 16#7190;
   // UNICODE_TO_GBK[19643] := 16#9FC7;
   // UNICODE_TO_GBK[19644] := 16#7191;
   // UNICODE_TO_GBK[19645] := 16#9FC8;
   // UNICODE_TO_GBK[19646] := 16#7192;
   // UNICODE_TO_GBK[19647] := 16#9FC9;
   // UNICODE_TO_GBK[19648] := 16#7193;
   // UNICODE_TO_GBK[19649] := 16#9FCA;
   // UNICODE_TO_GBK[19650] := 16#7194;
   // UNICODE_TO_GBK[19651] := 16#C8DB;
   // UNICODE_TO_GBK[19652] := 16#7195;
   // UNICODE_TO_GBK[19653] := 16#9FCB;
   // UNICODE_TO_GBK[19654] := 16#7196;
   // UNICODE_TO_GBK[19655] := 16#9FCC;
   // UNICODE_TO_GBK[19656] := 16#7197;
   // UNICODE_TO_GBK[19657] := 16#9FCD;
   // UNICODE_TO_GBK[19658] := 16#7198;
   // UNICODE_TO_GBK[19659] := 16#ECD6;
   // UNICODE_TO_GBK[19660] := 16#7199;
   // UNICODE_TO_GBK[19661] := 16#CEF5;
   // UNICODE_TO_GBK[19662] := 16#719A;
   // UNICODE_TO_GBK[19663] := 16#9FCE;
   // UNICODE_TO_GBK[19664] := 16#719B;
   // UNICODE_TO_GBK[19665] := 16#9FCF;
   // UNICODE_TO_GBK[19666] := 16#719C;
   // UNICODE_TO_GBK[19667] := 16#9FD0;
   // UNICODE_TO_GBK[19668] := 16#719D;
   // UNICODE_TO_GBK[19669] := 16#9FD1;
   // UNICODE_TO_GBK[19670] := 16#719E;
   // UNICODE_TO_GBK[19671] := 16#9FD2;
   // UNICODE_TO_GBK[19672] := 16#719F;
   // UNICODE_TO_GBK[19673] := 16#CAEC;
   // UNICODE_TO_GBK[19674] := 16#71A0;
   // UNICODE_TO_GBK[19675] := 16#ECDA;
   // UNICODE_TO_GBK[19676] := 16#71A1;
   // UNICODE_TO_GBK[19677] := 16#9FD3;
   // UNICODE_TO_GBK[19678] := 16#71A2;
   // UNICODE_TO_GBK[19679] := 16#9FD4;
   // UNICODE_TO_GBK[19680] := 16#71A3;
   // UNICODE_TO_GBK[19681] := 16#9FD5;
   // UNICODE_TO_GBK[19682] := 16#71A4;
   // UNICODE_TO_GBK[19683] := 16#9FD6;
   // UNICODE_TO_GBK[19684] := 16#71A5;
   // UNICODE_TO_GBK[19685] := 16#9FD7;
   // UNICODE_TO_GBK[19686] := 16#71A6;
   // UNICODE_TO_GBK[19687] := 16#9FD8;
   // UNICODE_TO_GBK[19688] := 16#71A7;
   // UNICODE_TO_GBK[19689] := 16#9FD9;
   // UNICODE_TO_GBK[19690] := 16#71A8;
   // UNICODE_TO_GBK[19691] := 16#ECD9;
   // UNICODE_TO_GBK[19692] := 16#71A9;
   // UNICODE_TO_GBK[19693] := 16#9FDA;
   // UNICODE_TO_GBK[19694] := 16#71AA;
   // UNICODE_TO_GBK[19695] := 16#9FDB;
   // UNICODE_TO_GBK[19696] := 16#71AB;
   // UNICODE_TO_GBK[19697] := 16#9FDC;
   // UNICODE_TO_GBK[19698] := 16#71AC;
   // UNICODE_TO_GBK[19699] := 16#B0BE;
   // UNICODE_TO_GBK[19700] := 16#71AD;
   // UNICODE_TO_GBK[19701] := 16#9FDD;
   // UNICODE_TO_GBK[19702] := 16#71AE;
   // UNICODE_TO_GBK[19703] := 16#9FDE;
   // UNICODE_TO_GBK[19704] := 16#71AF;
   // UNICODE_TO_GBK[19705] := 16#9FDF;
   // UNICODE_TO_GBK[19706] := 16#71B0;
   // UNICODE_TO_GBK[19707] := 16#9FE0;
   // UNICODE_TO_GBK[19708] := 16#71B1;
   // UNICODE_TO_GBK[19709] := 16#9FE1;
   // UNICODE_TO_GBK[19710] := 16#71B2;
   // UNICODE_TO_GBK[19711] := 16#9FE2;
   // UNICODE_TO_GBK[19712] := 16#71B3;
   // UNICODE_TO_GBK[19713] := 16#ECD7;
   // UNICODE_TO_GBK[19714] := 16#71B4;
   // UNICODE_TO_GBK[19715] := 16#9FE3;
   // UNICODE_TO_GBK[19716] := 16#71B5;
   // UNICODE_TO_GBK[19717] := 16#ECD8;
   // UNICODE_TO_GBK[19718] := 16#71B6;
   // UNICODE_TO_GBK[19719] := 16#9FE4;
   // UNICODE_TO_GBK[19720] := 16#71B7;
   // UNICODE_TO_GBK[19721] := 16#9FE5;
   // UNICODE_TO_GBK[19722] := 16#71B8;
   // UNICODE_TO_GBK[19723] := 16#9FE6;
   // UNICODE_TO_GBK[19724] := 16#71B9;
   // UNICODE_TO_GBK[19725] := 16#ECE4;
   // UNICODE_TO_GBK[19726] := 16#71BA;
   // UNICODE_TO_GBK[19727] := 16#9FE7;
   // UNICODE_TO_GBK[19728] := 16#71BB;
   // UNICODE_TO_GBK[19729] := 16#9FE8;
   // UNICODE_TO_GBK[19730] := 16#71BC;
   // UNICODE_TO_GBK[19731] := 16#9FE9;
   // UNICODE_TO_GBK[19732] := 16#71BD;
   // UNICODE_TO_GBK[19733] := 16#9FEA;
   // UNICODE_TO_GBK[19734] := 16#71BE;
   // UNICODE_TO_GBK[19735] := 16#9FEB;
   // UNICODE_TO_GBK[19736] := 16#71BF;
   // UNICODE_TO_GBK[19737] := 16#9FEC;
   // UNICODE_TO_GBK[19738] := 16#71C0;
   // UNICODE_TO_GBK[19739] := 16#9FED;
   // UNICODE_TO_GBK[19740] := 16#71C1;
   // UNICODE_TO_GBK[19741] := 16#9FEE;
   // UNICODE_TO_GBK[19742] := 16#71C2;
   // UNICODE_TO_GBK[19743] := 16#9FEF;
   // UNICODE_TO_GBK[19744] := 16#71C3;
   // UNICODE_TO_GBK[19745] := 16#C8BC;
   // UNICODE_TO_GBK[19746] := 16#71C4;
   // UNICODE_TO_GBK[19747] := 16#9FF0;
   // UNICODE_TO_GBK[19748] := 16#71C5;
   // UNICODE_TO_GBK[19749] := 16#9FF1;
   // UNICODE_TO_GBK[19750] := 16#71C6;
   // UNICODE_TO_GBK[19751] := 16#9FF2;
   // UNICODE_TO_GBK[19752] := 16#71C7;
   // UNICODE_TO_GBK[19753] := 16#9FF3;
   // UNICODE_TO_GBK[19754] := 16#71C8;
   // UNICODE_TO_GBK[19755] := 16#9FF4;
   // UNICODE_TO_GBK[19756] := 16#71C9;
   // UNICODE_TO_GBK[19757] := 16#9FF5;
   // UNICODE_TO_GBK[19758] := 16#71CA;
   // UNICODE_TO_GBK[19759] := 16#9FF6;
   // UNICODE_TO_GBK[19760] := 16#71CB;
   // UNICODE_TO_GBK[19761] := 16#9FF7;
   // UNICODE_TO_GBK[19762] := 16#71CC;
   // UNICODE_TO_GBK[19763] := 16#9FF8;
   // UNICODE_TO_GBK[19764] := 16#71CD;
   // UNICODE_TO_GBK[19765] := 16#9FF9;
   // UNICODE_TO_GBK[19766] := 16#71CE;
   // UNICODE_TO_GBK[19767] := 16#C1C7;
   // UNICODE_TO_GBK[19768] := 16#71CF;
   // UNICODE_TO_GBK[19769] := 16#9FFA;
   // UNICODE_TO_GBK[19770] := 16#71D0;
   // UNICODE_TO_GBK[19771] := 16#9FFB;
   // UNICODE_TO_GBK[19772] := 16#71D1;
   // UNICODE_TO_GBK[19773] := 16#9FFC;
   // UNICODE_TO_GBK[19774] := 16#71D2;
   // UNICODE_TO_GBK[19775] := 16#9FFD;
   // UNICODE_TO_GBK[19776] := 16#71D3;
   // UNICODE_TO_GBK[19777] := 16#9FFE;
   // UNICODE_TO_GBK[19778] := 16#71D4;
   // UNICODE_TO_GBK[19779] := 16#ECDC;
   // UNICODE_TO_GBK[19780] := 16#71D5;
   // UNICODE_TO_GBK[19781] := 16#D1E0;
   // UNICODE_TO_GBK[19782] := 16#71D6;
   // UNICODE_TO_GBK[19783] := 16#A040;
   // UNICODE_TO_GBK[19784] := 16#71D7;
   // UNICODE_TO_GBK[19785] := 16#A041;
   // UNICODE_TO_GBK[19786] := 16#71D8;
   // UNICODE_TO_GBK[19787] := 16#A042;
   // UNICODE_TO_GBK[19788] := 16#71D9;
   // UNICODE_TO_GBK[19789] := 16#A043;
   // UNICODE_TO_GBK[19790] := 16#71DA;
   // UNICODE_TO_GBK[19791] := 16#A044;
   // UNICODE_TO_GBK[19792] := 16#71DB;
   // UNICODE_TO_GBK[19793] := 16#A045;
   // UNICODE_TO_GBK[19794] := 16#71DC;
   // UNICODE_TO_GBK[19795] := 16#A046;
   // UNICODE_TO_GBK[19796] := 16#71DD;
   // UNICODE_TO_GBK[19797] := 16#A047;
   // UNICODE_TO_GBK[19798] := 16#71DE;
   // UNICODE_TO_GBK[19799] := 16#A048;
   // UNICODE_TO_GBK[19800] := 16#71DF;
   // UNICODE_TO_GBK[19801] := 16#A049;
   // UNICODE_TO_GBK[19802] := 16#71E0;
   // UNICODE_TO_GBK[19803] := 16#ECDB;
   // UNICODE_TO_GBK[19804] := 16#71E1;
   // UNICODE_TO_GBK[19805] := 16#A04A;
   // UNICODE_TO_GBK[19806] := 16#71E2;
   // UNICODE_TO_GBK[19807] := 16#A04B;
   // UNICODE_TO_GBK[19808] := 16#71E3;
   // UNICODE_TO_GBK[19809] := 16#A04C;
   // UNICODE_TO_GBK[19810] := 16#71E4;
   // UNICODE_TO_GBK[19811] := 16#A04D;
   // UNICODE_TO_GBK[19812] := 16#71E5;
   // UNICODE_TO_GBK[19813] := 16#D4EF;
   // UNICODE_TO_GBK[19814] := 16#71E6;
   // UNICODE_TO_GBK[19815] := 16#A04E;
   // UNICODE_TO_GBK[19816] := 16#71E7;
   // UNICODE_TO_GBK[19817] := 16#ECDD;
   // UNICODE_TO_GBK[19818] := 16#71E8;
   // UNICODE_TO_GBK[19819] := 16#A04F;
   // UNICODE_TO_GBK[19820] := 16#71E9;
   // UNICODE_TO_GBK[19821] := 16#A050;
   // UNICODE_TO_GBK[19822] := 16#71EA;
   // UNICODE_TO_GBK[19823] := 16#A051;
   // UNICODE_TO_GBK[19824] := 16#71EB;
   // UNICODE_TO_GBK[19825] := 16#A052;
